// TIA Portal V21 export
FUNCTION "ALARMS PRINT" : Void   // FC2, LAD
{ S7_Optimized_Access := 'TRUE' }
// stored: SetENOAutomatically false
   VAR_TEMP   // added for the SCL form of the ladder/FBD networks
      _w1 : Bool;
      _w2 : Bool;
   END_VAR
BEGIN

REGION Network 1
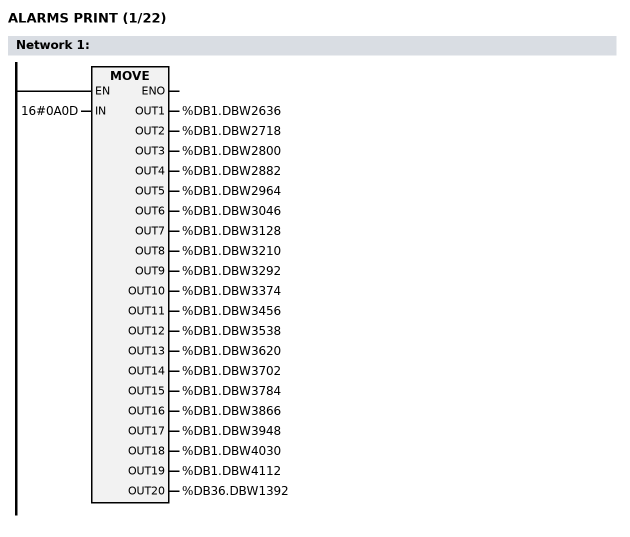
   RUNG wire#powerrail
      Move(in := 16#0A0D, out1 => %DB1.DBW2636, out2 => %DB1.DBW2718, out3 => %DB1.DBW2800, out4 => %DB1.DBW2882, out5 => %DB1.DBW2964, out6 => %DB1.DBW3046, out7 => %DB1.DBW3128, out8 => %DB1.DBW3210, out9 => %DB1.DBW3292, out10 => %DB1.DBW3374, out11 => %DB1.DBW3456, out12 => %DB1.DBW3538, out13 => %DB1.DBW3620, out14 => %DB1.DBW3702, out15 => %DB1.DBW3784, out16 => %DB1.DBW3866, out17 => %DB1.DBW3948, out18 => %DB1.DBW4030, out19 => %DB1.DBW4112, out20 => %DB36.DBW1392)
   END_RUNG
   // the same network as SCL:
   %DB1.DBW2636 := 16#0A0D;
   %DB1.DBW2718 := 16#0A0D;
   %DB1.DBW2800 := 16#0A0D;
   %DB1.DBW2882 := 16#0A0D;
   %DB1.DBW2964 := 16#0A0D;
   %DB1.DBW3046 := 16#0A0D;
   %DB1.DBW3128 := 16#0A0D;
   %DB1.DBW3210 := 16#0A0D;
   %DB1.DBW3292 := 16#0A0D;
   %DB1.DBW3374 := 16#0A0D;
   %DB1.DBW3456 := 16#0A0D;
   %DB1.DBW3538 := 16#0A0D;
   %DB1.DBW3620 := 16#0A0D;
   %DB1.DBW3702 := 16#0A0D;
   %DB1.DBW3784 := 16#0A0D;
   %DB1.DBW3866 := 16#0A0D;
   %DB1.DBW3948 := 16#0A0D;
   %DB1.DBW4030 := 16#0A0D;
   %DB1.DBW4112 := 16#0A0D;
   %DB36.DBW1392 := 16#0A0D;
END_REGION

REGION Network 2
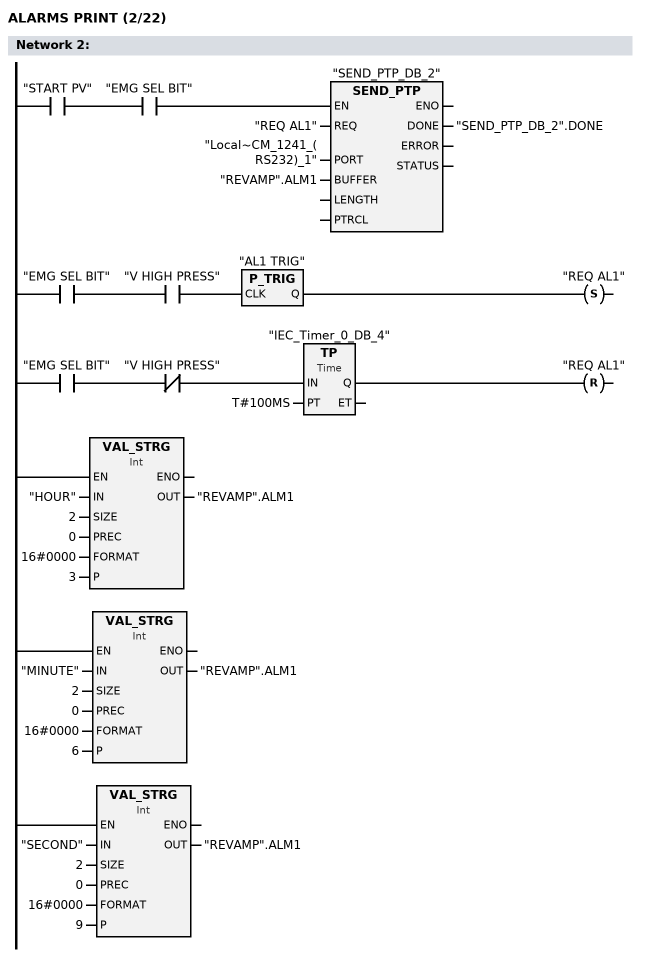
   RUNG wire#powerrail
      Contact( "START PV" )
      Contact( "EMG SEL BIT" )
      "SEND_PTP_DB_2".SEND_PTP(REQ := "REQ AL1", PORT := "Local~CM_1241_(RS232)_1", BUFFER := "REVAMP".ALM1, LENGTH :=, PTRCL :=, DONE => "SEND_PTP_DB_2".DONE, ERROR =>, STATUS =>)
   END_RUNG
   RUNG wire#powerrail
      Contact( "EMG SEL BIT" )
      Contact( "V HIGH PRESS" )
      P_Trig( "AL1 TRIG" )
      S_Coil( "REQ AL1" )
   END_RUNG
   RUNG wire#powerrail
      Contact( "EMG SEL BIT" )
      I_Contact( "V HIGH PRESS" )
      { S7_Templates := "time_type := Time" } "IEC_Timer_0_DB_4".TP(pt := T#100MS, et =>)
      R_Coil( "REQ AL1" )
   END_RUNG
   RUNG wire#powerrail
      { S7_Templates := "[value_type := Int, str_type := String]" } VAL_STRG(IN := "HOUR", SIZE := 2, PREC := 0, FORMAT := 16#0000, P := 3, OUT => "REVAMP".ALM1)
   END_RUNG
   RUNG wire#powerrail
      { S7_Templates := "[value_type := Int, str_type := String]" } VAL_STRG(IN := "MINUTE", SIZE := 2, PREC := 0, FORMAT := 16#0000, P := 6, OUT => "REVAMP".ALM1)
   END_RUNG
   RUNG wire#powerrail
      { S7_Templates := "[value_type := Int, str_type := String]" } VAL_STRG(IN := "SECOND", SIZE := 2, PREC := 0, FORMAT := 16#0000, P := 9, OUT => "REVAMP".ALM1)
   END_RUNG
   // the same network as SCL:
   IF "START PV" AND "EMG SEL BIT" THEN
       "SEND_PTP_DB_2"(REQ := "REQ AL1",   // SEND_PTP
                       PORT := "Local~CM_1241_(RS232)_1",
                       BUFFER := "REVAMP".ALM1,
                       DONE => "SEND_PTP_DB_2".DONE);
   END_IF;
   #_w1 := "EMG SEL BIT" AND "V HIGH PRESS";
   #_w2 := #_w1 AND NOT "AL1 TRIG";   // rising edge
   "AL1 TRIG" := #_w1;
   IF #_w2 THEN "REQ AL1" := TRUE; END_IF;
   "IEC_Timer_0_DB_4".TP(IN := "EMG SEL BIT" AND NOT "V HIGH PRESS", PT := T#100MS);
   IF "IEC_Timer_0_DB_4".Q THEN "REQ AL1" := FALSE; END_IF;
   VAL_STRG(IN := "HOUR", SIZE := 2, PREC := 0, FORMAT := 16#0000, P := 3, OUT => "REVAMP".ALM1);
   VAL_STRG(IN := "MINUTE", SIZE := 2, PREC := 0, FORMAT := 16#0000, P := 6, OUT => "REVAMP".ALM1);
   VAL_STRG(IN := "SECOND", SIZE := 2, PREC := 0, FORMAT := 16#0000, P := 9, OUT => "REVAMP".ALM1);
END_REGION

REGION Network 3
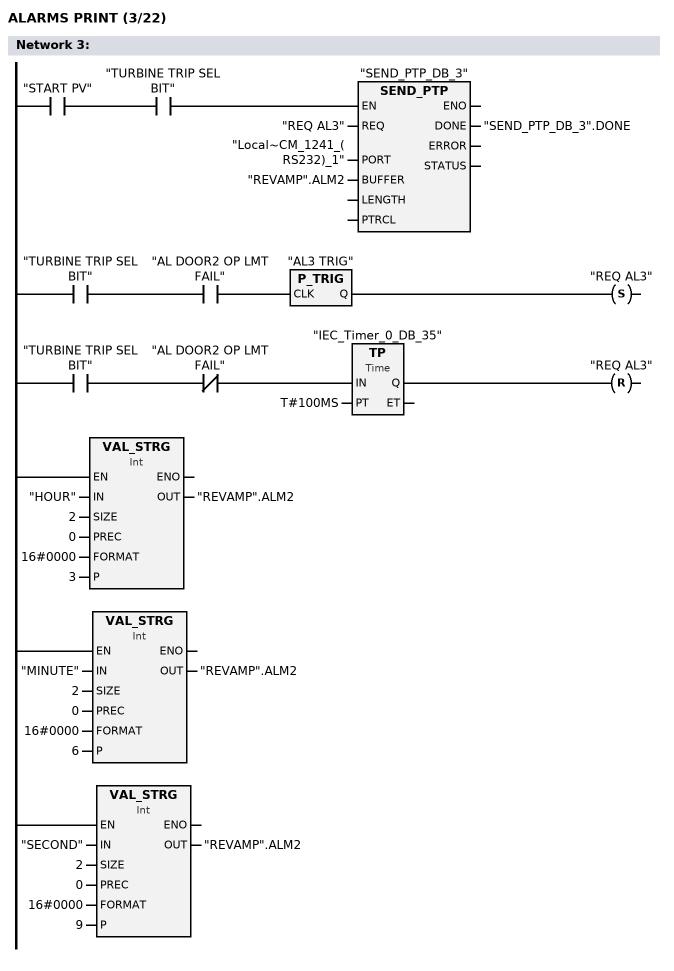
   RUNG wire#powerrail
      Contact( "START PV" )
      Contact( "TURBINE TRIP SEL BIT" )
      "SEND_PTP_DB_3".SEND_PTP(REQ := "REQ AL3", PORT := "Local~CM_1241_(RS232)_1", BUFFER := "REVAMP".ALM2, LENGTH :=, PTRCL :=, DONE => "SEND_PTP_DB_3".DONE, ERROR =>, STATUS =>)
   END_RUNG
   RUNG wire#powerrail
      Contact( "TURBINE TRIP SEL BIT" )
      Contact( "AL DOOR2 OP LMT FAIL" )
      P_Trig( "AL3 TRIG" )
      S_Coil( "REQ AL3" )
   END_RUNG
   RUNG wire#powerrail
      Contact( "TURBINE TRIP SEL BIT" )
      I_Contact( "AL DOOR2 OP LMT FAIL" )
      { S7_Templates := "time_type := Time" } "IEC_Timer_0_DB_35".TP(pt := T#100MS, et =>)
      R_Coil( "REQ AL3" )
   END_RUNG
   RUNG wire#powerrail
      { S7_Templates := "[value_type := Int, str_type := String]" } VAL_STRG(IN := "HOUR", SIZE := 2, PREC := 0, FORMAT := 16#0000, P := 3, OUT => "REVAMP".ALM2)
   END_RUNG
   RUNG wire#powerrail
      { S7_Templates := "[value_type := Int, str_type := String]" } VAL_STRG(IN := "MINUTE", SIZE := 2, PREC := 0, FORMAT := 16#0000, P := 6, OUT => "REVAMP".ALM2)
   END_RUNG
   RUNG wire#powerrail
      { S7_Templates := "[value_type := Int, str_type := String]" } VAL_STRG(IN := "SECOND", SIZE := 2, PREC := 0, FORMAT := 16#0000, P := 9, OUT => "REVAMP".ALM2)
   END_RUNG
   // the same network as SCL:
   IF "START PV" AND "TURBINE TRIP SEL BIT" THEN
       "SEND_PTP_DB_3"(REQ := "REQ AL3",   // SEND_PTP
                       PORT := "Local~CM_1241_(RS232)_1",
                       BUFFER := "REVAMP".ALM2,
                       DONE => "SEND_PTP_DB_3".DONE);
   END_IF;
   #_w1 := "TURBINE TRIP SEL BIT" AND "AL DOOR2 OP LMT FAIL";
   #_w2 := #_w1 AND NOT "AL3 TRIG";   // rising edge
   "AL3 TRIG" := #_w1;
   IF #_w2 THEN "REQ AL3" := TRUE; END_IF;
   "IEC_Timer_0_DB_35".TP(IN := "TURBINE TRIP SEL BIT" AND NOT "AL DOOR2 OP LMT FAIL", PT := T#100MS);
   IF "IEC_Timer_0_DB_35".Q THEN "REQ AL3" := FALSE; END_IF;
   VAL_STRG(IN := "HOUR", SIZE := 2, PREC := 0, FORMAT := 16#0000, P := 3, OUT => "REVAMP".ALM2);
   VAL_STRG(IN := "MINUTE", SIZE := 2, PREC := 0, FORMAT := 16#0000, P := 6, OUT => "REVAMP".ALM2);
   VAL_STRG(IN := "SECOND", SIZE := 2, PREC := 0, FORMAT := 16#0000, P := 9, OUT => "REVAMP".ALM2);
END_REGION

REGION Network 4
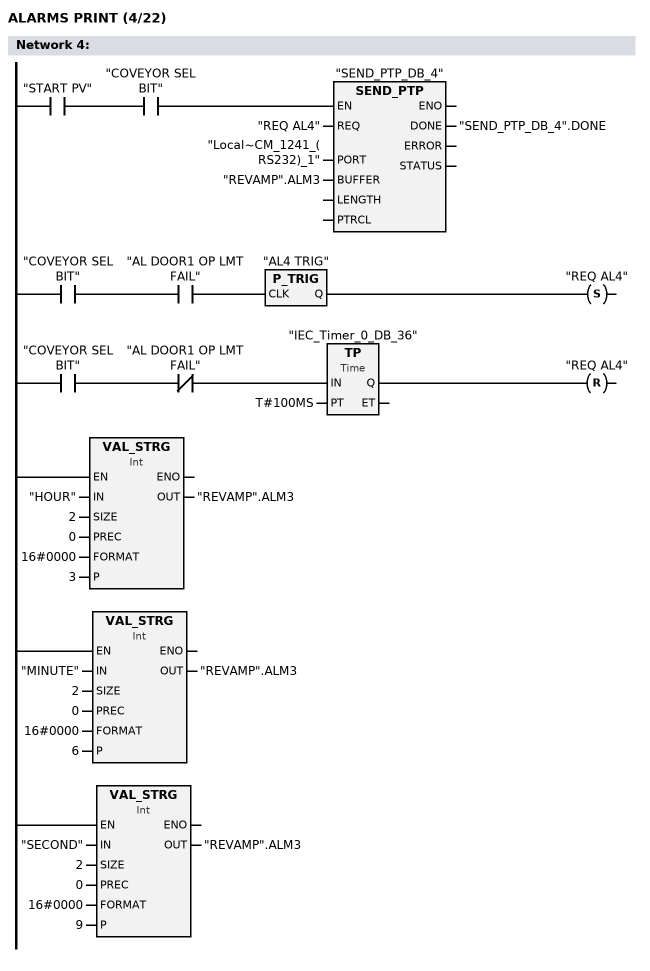
   RUNG wire#powerrail
      Contact( "START PV" )
      Contact( "COVEYOR SEL BIT" )
      "SEND_PTP_DB_4".SEND_PTP(REQ := "REQ AL4", PORT := "Local~CM_1241_(RS232)_1", BUFFER := "REVAMP".ALM3, LENGTH :=, PTRCL :=, DONE => "SEND_PTP_DB_4".DONE, ERROR =>, STATUS =>)
   END_RUNG
   RUNG wire#powerrail
      Contact( "COVEYOR SEL BIT" )
      Contact( "AL DOOR1 OP LMT FAIL" )
      P_Trig( "AL4 TRIG" )
      S_Coil( "REQ AL4" )
   END_RUNG
   RUNG wire#powerrail
      Contact( "COVEYOR SEL BIT" )
      I_Contact( "AL DOOR1 OP LMT FAIL" )
      { S7_Templates := "time_type := Time" } "IEC_Timer_0_DB_36".TP(pt := T#100MS, et =>)
      R_Coil( "REQ AL4" )
   END_RUNG
   RUNG wire#powerrail
      { S7_Templates := "[value_type := Int, str_type := String]" } VAL_STRG(IN := "HOUR", SIZE := 2, PREC := 0, FORMAT := 16#0000, P := 3, OUT => "REVAMP".ALM3)
   END_RUNG
   RUNG wire#powerrail
      { S7_Templates := "[value_type := Int, str_type := String]" } VAL_STRG(IN := "MINUTE", SIZE := 2, PREC := 0, FORMAT := 16#0000, P := 6, OUT => "REVAMP".ALM3)
   END_RUNG
   RUNG wire#powerrail
      { S7_Templates := "[value_type := Int, str_type := String]" } VAL_STRG(IN := "SECOND", SIZE := 2, PREC := 0, FORMAT := 16#0000, P := 9, OUT => "REVAMP".ALM3)
   END_RUNG
   // the same network as SCL:
   IF "START PV" AND "COVEYOR SEL BIT" THEN
       "SEND_PTP_DB_4"(REQ := "REQ AL4",   // SEND_PTP
                       PORT := "Local~CM_1241_(RS232)_1",
                       BUFFER := "REVAMP".ALM3,
                       DONE => "SEND_PTP_DB_4".DONE);
   END_IF;
   #_w1 := "COVEYOR SEL BIT" AND "AL DOOR1 OP LMT FAIL";
   #_w2 := #_w1 AND NOT "AL4 TRIG";   // rising edge
   "AL4 TRIG" := #_w1;
   IF #_w2 THEN "REQ AL4" := TRUE; END_IF;
   "IEC_Timer_0_DB_36".TP(IN := "COVEYOR SEL BIT" AND NOT "AL DOOR1 OP LMT FAIL", PT := T#100MS);
   IF "IEC_Timer_0_DB_36".Q THEN "REQ AL4" := FALSE; END_IF;
   VAL_STRG(IN := "HOUR", SIZE := 2, PREC := 0, FORMAT := 16#0000, P := 3, OUT => "REVAMP".ALM3);
   VAL_STRG(IN := "MINUTE", SIZE := 2, PREC := 0, FORMAT := 16#0000, P := 6, OUT => "REVAMP".ALM3);
   VAL_STRG(IN := "SECOND", SIZE := 2, PREC := 0, FORMAT := 16#0000, P := 9, OUT => "REVAMP".ALM3);
END_REGION

REGION Network 5
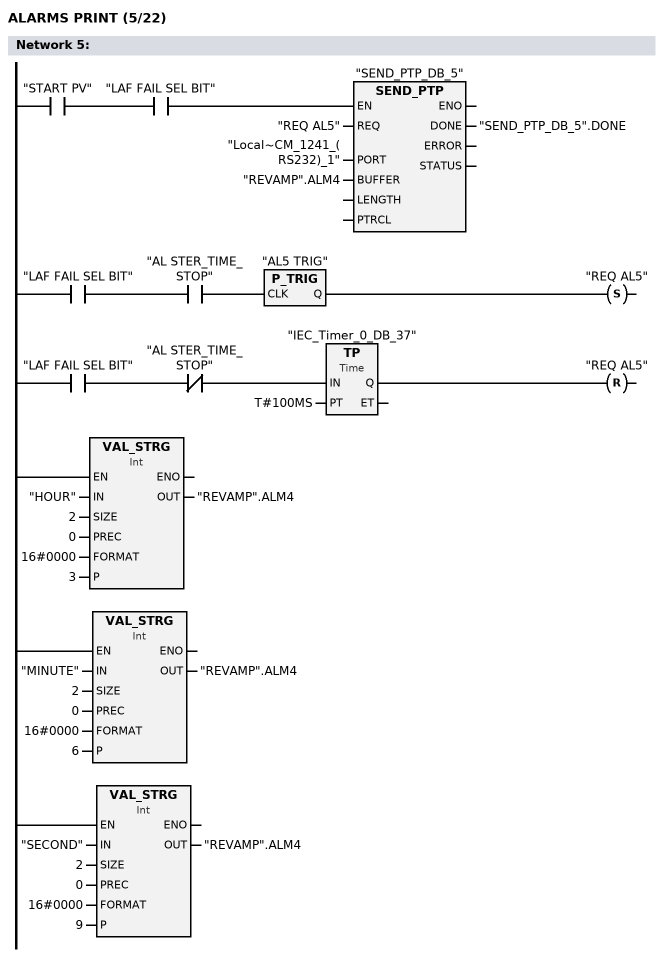
   RUNG wire#powerrail
      Contact( "START PV" )
      Contact( "LAF FAIL SEL BIT" )
      "SEND_PTP_DB_5".SEND_PTP(REQ := "REQ AL5", PORT := "Local~CM_1241_(RS232)_1", BUFFER := "REVAMP".ALM4, LENGTH :=, PTRCL :=, DONE => "SEND_PTP_DB_5".DONE, ERROR =>, STATUS =>)
   END_RUNG
   RUNG wire#powerrail
      Contact( "LAF FAIL SEL BIT" )
      Contact( "AL STER_TIME_STOP" )
      P_Trig( "AL5 TRIG" )
      S_Coil( "REQ AL5" )
   END_RUNG
   RUNG wire#powerrail
      Contact( "LAF FAIL SEL BIT" )
      I_Contact( "AL STER_TIME_STOP" )
      { S7_Templates := "time_type := Time" } "IEC_Timer_0_DB_37".TP(pt := T#100MS, et =>)
      R_Coil( "REQ AL5" )
   END_RUNG
   RUNG wire#powerrail
      { S7_Templates := "[value_type := Int, str_type := String]" } VAL_STRG(IN := "HOUR", SIZE := 2, PREC := 0, FORMAT := 16#0000, P := 3, OUT => "REVAMP".ALM4)
   END_RUNG
   RUNG wire#powerrail
      { S7_Templates := "[value_type := Int, str_type := String]" } VAL_STRG(IN := "MINUTE", SIZE := 2, PREC := 0, FORMAT := 16#0000, P := 6, OUT => "REVAMP".ALM4)
   END_RUNG
   RUNG wire#powerrail
      { S7_Templates := "[value_type := Int, str_type := String]" } VAL_STRG(IN := "SECOND", SIZE := 2, PREC := 0, FORMAT := 16#0000, P := 9, OUT => "REVAMP".ALM4)
   END_RUNG
   // the same network as SCL:
   IF "START PV" AND "LAF FAIL SEL BIT" THEN
       "SEND_PTP_DB_5"(REQ := "REQ AL5",   // SEND_PTP
                       PORT := "Local~CM_1241_(RS232)_1",
                       BUFFER := "REVAMP".ALM4,
                       DONE => "SEND_PTP_DB_5".DONE);
   END_IF;
   #_w1 := "LAF FAIL SEL BIT" AND "AL STER_TIME_STOP";
   #_w2 := #_w1 AND NOT "AL5 TRIG";   // rising edge
   "AL5 TRIG" := #_w1;
   IF #_w2 THEN "REQ AL5" := TRUE; END_IF;
   "IEC_Timer_0_DB_37".TP(IN := "LAF FAIL SEL BIT" AND NOT "AL STER_TIME_STOP", PT := T#100MS);
   IF "IEC_Timer_0_DB_37".Q THEN "REQ AL5" := FALSE; END_IF;
   VAL_STRG(IN := "HOUR", SIZE := 2, PREC := 0, FORMAT := 16#0000, P := 3, OUT => "REVAMP".ALM4);
   VAL_STRG(IN := "MINUTE", SIZE := 2, PREC := 0, FORMAT := 16#0000, P := 6, OUT => "REVAMP".ALM4);
   VAL_STRG(IN := "SECOND", SIZE := 2, PREC := 0, FORMAT := 16#0000, P := 9, OUT => "REVAMP".ALM4);
END_REGION

REGION Network 6
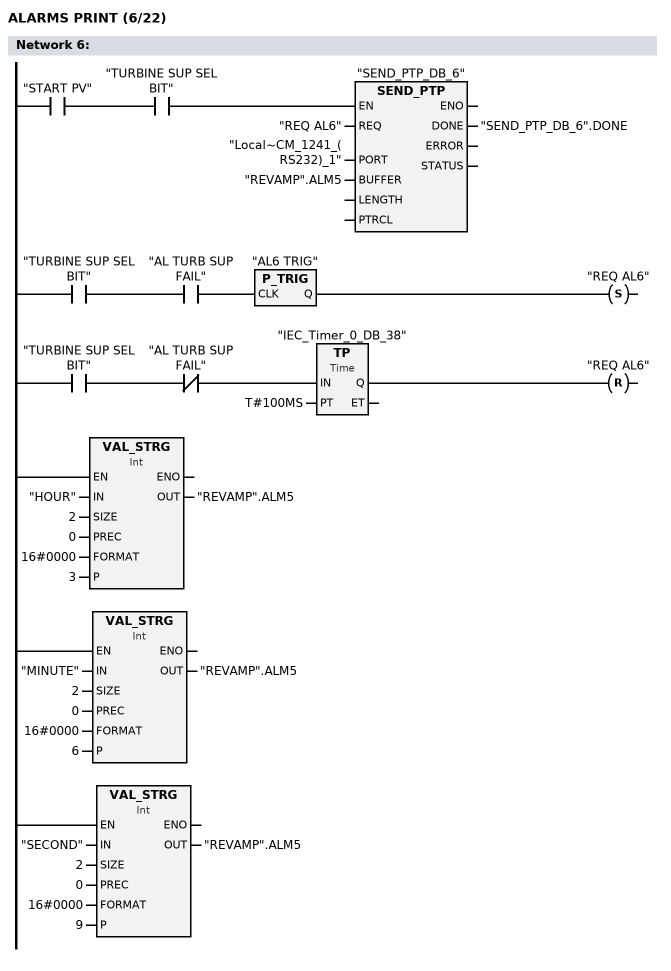
   RUNG wire#powerrail
      Contact( "START PV" )
      Contact( "TURBINE SUP SEL BIT" )
      "SEND_PTP_DB_6".SEND_PTP(REQ := "REQ AL6", PORT := "Local~CM_1241_(RS232)_1", BUFFER := "REVAMP".ALM5, LENGTH :=, PTRCL :=, DONE => "SEND_PTP_DB_6".DONE, ERROR =>, STATUS =>)
   END_RUNG
   RUNG wire#powerrail
      Contact( "TURBINE SUP SEL BIT" )
      Contact( "AL TURB SUP FAIL" )
      P_Trig( "AL6 TRIG" )
      S_Coil( "REQ AL6" )
   END_RUNG
   RUNG wire#powerrail
      Contact( "TURBINE SUP SEL BIT" )
      I_Contact( "AL TURB SUP FAIL" )
      { S7_Templates := "time_type := Time" } "IEC_Timer_0_DB_38".TP(pt := T#100MS, et =>)
      R_Coil( "REQ AL6" )
   END_RUNG
   RUNG wire#powerrail
      { S7_Templates := "[value_type := Int, str_type := String]" } VAL_STRG(IN := "HOUR", SIZE := 2, PREC := 0, FORMAT := 16#0000, P := 3, OUT => "REVAMP".ALM5)
   END_RUNG
   RUNG wire#powerrail
      { S7_Templates := "[value_type := Int, str_type := String]" } VAL_STRG(IN := "MINUTE", SIZE := 2, PREC := 0, FORMAT := 16#0000, P := 6, OUT => "REVAMP".ALM5)
   END_RUNG
   RUNG wire#powerrail
      { S7_Templates := "[value_type := Int, str_type := String]" } VAL_STRG(IN := "SECOND", SIZE := 2, PREC := 0, FORMAT := 16#0000, P := 9, OUT => "REVAMP".ALM5)
   END_RUNG
   // the same network as SCL:
   IF "START PV" AND "TURBINE SUP SEL BIT" THEN
       "SEND_PTP_DB_6"(REQ := "REQ AL6",   // SEND_PTP
                       PORT := "Local~CM_1241_(RS232)_1",
                       BUFFER := "REVAMP".ALM5,
                       DONE => "SEND_PTP_DB_6".DONE);
   END_IF;
   #_w1 := "TURBINE SUP SEL BIT" AND "AL TURB SUP FAIL";
   #_w2 := #_w1 AND NOT "AL6 TRIG";   // rising edge
   "AL6 TRIG" := #_w1;
   IF #_w2 THEN "REQ AL6" := TRUE; END_IF;
   "IEC_Timer_0_DB_38".TP(IN := "TURBINE SUP SEL BIT" AND NOT "AL TURB SUP FAIL", PT := T#100MS);
   IF "IEC_Timer_0_DB_38".Q THEN "REQ AL6" := FALSE; END_IF;
   VAL_STRG(IN := "HOUR", SIZE := 2, PREC := 0, FORMAT := 16#0000, P := 3, OUT => "REVAMP".ALM5);
   VAL_STRG(IN := "MINUTE", SIZE := 2, PREC := 0, FORMAT := 16#0000, P := 6, OUT => "REVAMP".ALM5);
   VAL_STRG(IN := "SECOND", SIZE := 2, PREC := 0, FORMAT := 16#0000, P := 9, OUT => "REVAMP".ALM5);
END_REGION

REGION Network 7
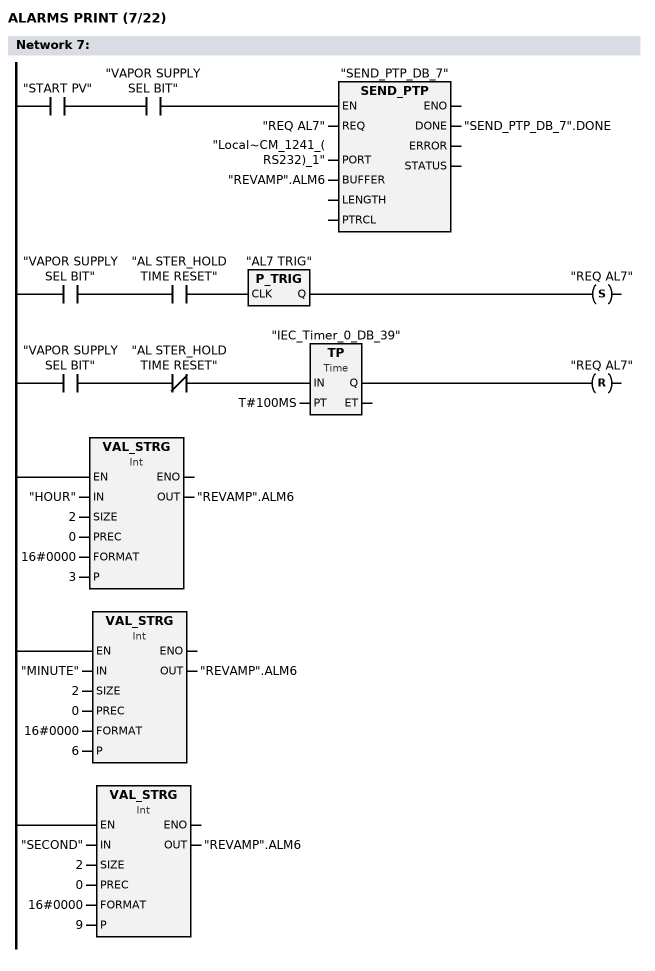
   RUNG wire#powerrail
      Contact( "START PV" )
      Contact( "VAPOR SUPPLY SEL BIT" )
      "SEND_PTP_DB_7".SEND_PTP(REQ := "REQ AL7", PORT := "Local~CM_1241_(RS232)_1", BUFFER := "REVAMP".ALM6, LENGTH :=, PTRCL :=, DONE => "SEND_PTP_DB_7".DONE, ERROR =>, STATUS =>)
   END_RUNG
   RUNG wire#powerrail
      Contact( "VAPOR SUPPLY SEL BIT" )
      Contact( "AL STER_HOLD TIME RESET" )
      P_Trig( "AL7 TRIG" )
      S_Coil( "REQ AL7" )
   END_RUNG
   RUNG wire#powerrail
      Contact( "VAPOR SUPPLY SEL BIT" )
      I_Contact( "AL STER_HOLD TIME RESET" )
      { S7_Templates := "time_type := Time" } "IEC_Timer_0_DB_39".TP(pt := T#100MS, et =>)
      R_Coil( "REQ AL7" )
   END_RUNG
   RUNG wire#powerrail
      { S7_Templates := "[value_type := Int, str_type := String]" } VAL_STRG(IN := "HOUR", SIZE := 2, PREC := 0, FORMAT := 16#0000, P := 3, OUT => "REVAMP".ALM6)
   END_RUNG
   RUNG wire#powerrail
      { S7_Templates := "[value_type := Int, str_type := String]" } VAL_STRG(IN := "MINUTE", SIZE := 2, PREC := 0, FORMAT := 16#0000, P := 6, OUT => "REVAMP".ALM6)
   END_RUNG
   RUNG wire#powerrail
      { S7_Templates := "[value_type := Int, str_type := String]" } VAL_STRG(IN := "SECOND", SIZE := 2, PREC := 0, FORMAT := 16#0000, P := 9, OUT => "REVAMP".ALM6)
   END_RUNG
   // the same network as SCL:
   IF "START PV" AND "VAPOR SUPPLY SEL BIT" THEN
       "SEND_PTP_DB_7"(REQ := "REQ AL7",   // SEND_PTP
                       PORT := "Local~CM_1241_(RS232)_1",
                       BUFFER := "REVAMP".ALM6,
                       DONE => "SEND_PTP_DB_7".DONE);
   END_IF;
   #_w1 := "VAPOR SUPPLY SEL BIT" AND "AL STER_HOLD TIME RESET";
   #_w2 := #_w1 AND NOT "AL7 TRIG";   // rising edge
   "AL7 TRIG" := #_w1;
   IF #_w2 THEN "REQ AL7" := TRUE; END_IF;
   "IEC_Timer_0_DB_39".TP(IN := "VAPOR SUPPLY SEL BIT" AND NOT "AL STER_HOLD TIME RESET", PT := T#100MS);
   IF "IEC_Timer_0_DB_39".Q THEN "REQ AL7" := FALSE; END_IF;
   VAL_STRG(IN := "HOUR", SIZE := 2, PREC := 0, FORMAT := 16#0000, P := 3, OUT => "REVAMP".ALM6);
   VAL_STRG(IN := "MINUTE", SIZE := 2, PREC := 0, FORMAT := 16#0000, P := 6, OUT => "REVAMP".ALM6);
   VAL_STRG(IN := "SECOND", SIZE := 2, PREC := 0, FORMAT := 16#0000, P := 9, OUT => "REVAMP".ALM6);
END_REGION

REGION Network 8
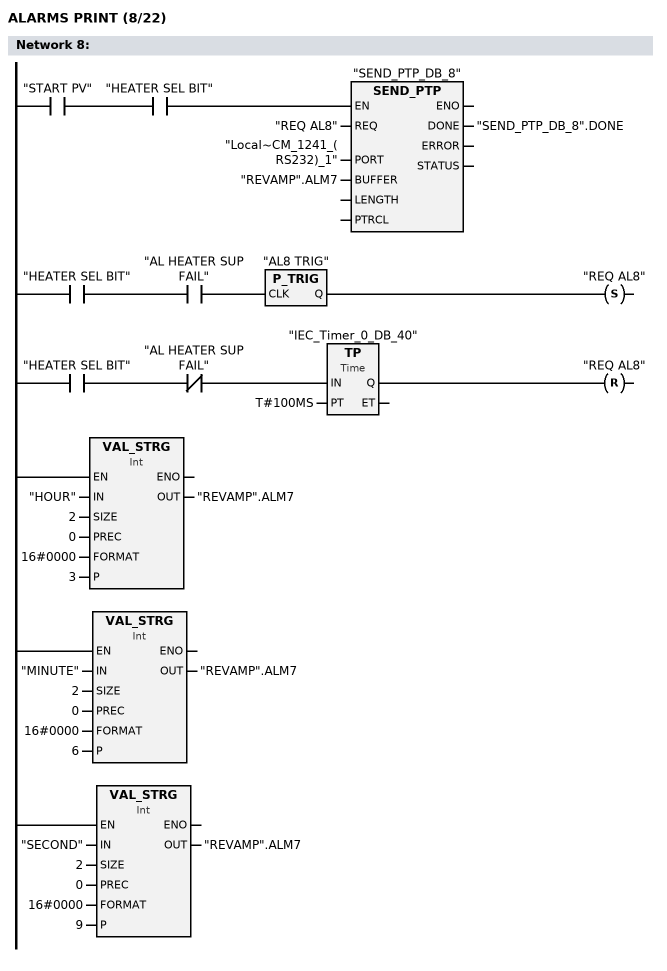
   RUNG wire#powerrail
      Contact( "START PV" )
      Contact( "HEATER SEL BIT" )
      "SEND_PTP_DB_8".SEND_PTP(REQ := "REQ AL8", PORT := "Local~CM_1241_(RS232)_1", BUFFER := "REVAMP".ALM7, LENGTH :=, PTRCL :=, DONE => "SEND_PTP_DB_8".DONE, ERROR =>, STATUS =>)
   END_RUNG
   RUNG wire#powerrail
      Contact( "HEATER SEL BIT" )
      Contact( "AL HEATER SUP FAIL" )
      P_Trig( "AL8 TRIG" )
      S_Coil( "REQ AL8" )
   END_RUNG
   RUNG wire#powerrail
      Contact( "HEATER SEL BIT" )
      I_Contact( "AL HEATER SUP FAIL" )
      { S7_Templates := "time_type := Time" } "IEC_Timer_0_DB_40".TP(pt := T#100MS, et =>)
      R_Coil( "REQ AL8" )
   END_RUNG
   RUNG wire#powerrail
      { S7_Templates := "[value_type := Int, str_type := String]" } VAL_STRG(IN := "HOUR", SIZE := 2, PREC := 0, FORMAT := 16#0000, P := 3, OUT => "REVAMP".ALM7)
   END_RUNG
   RUNG wire#powerrail
      { S7_Templates := "[value_type := Int, str_type := String]" } VAL_STRG(IN := "MINUTE", SIZE := 2, PREC := 0, FORMAT := 16#0000, P := 6, OUT => "REVAMP".ALM7)
   END_RUNG
   RUNG wire#powerrail
      { S7_Templates := "[value_type := Int, str_type := String]" } VAL_STRG(IN := "SECOND", SIZE := 2, PREC := 0, FORMAT := 16#0000, P := 9, OUT => "REVAMP".ALM7)
   END_RUNG
   // the same network as SCL:
   IF "START PV" AND "HEATER SEL BIT" THEN
       "SEND_PTP_DB_8"(REQ := "REQ AL8",   // SEND_PTP
                       PORT := "Local~CM_1241_(RS232)_1",
                       BUFFER := "REVAMP".ALM7,
                       DONE => "SEND_PTP_DB_8".DONE);
   END_IF;
   #_w1 := "HEATER SEL BIT" AND "AL HEATER SUP FAIL";
   #_w2 := #_w1 AND NOT "AL8 TRIG";   // rising edge
   "AL8 TRIG" := #_w1;
   IF #_w2 THEN "REQ AL8" := TRUE; END_IF;
   "IEC_Timer_0_DB_40".TP(IN := "HEATER SEL BIT" AND NOT "AL HEATER SUP FAIL", PT := T#100MS);
   IF "IEC_Timer_0_DB_40".Q THEN "REQ AL8" := FALSE; END_IF;
   VAL_STRG(IN := "HOUR", SIZE := 2, PREC := 0, FORMAT := 16#0000, P := 3, OUT => "REVAMP".ALM7);
   VAL_STRG(IN := "MINUTE", SIZE := 2, PREC := 0, FORMAT := 16#0000, P := 6, OUT => "REVAMP".ALM7);
   VAL_STRG(IN := "SECOND", SIZE := 2, PREC := 0, FORMAT := 16#0000, P := 9, OUT => "REVAMP".ALM7);
END_REGION

REGION Network 9
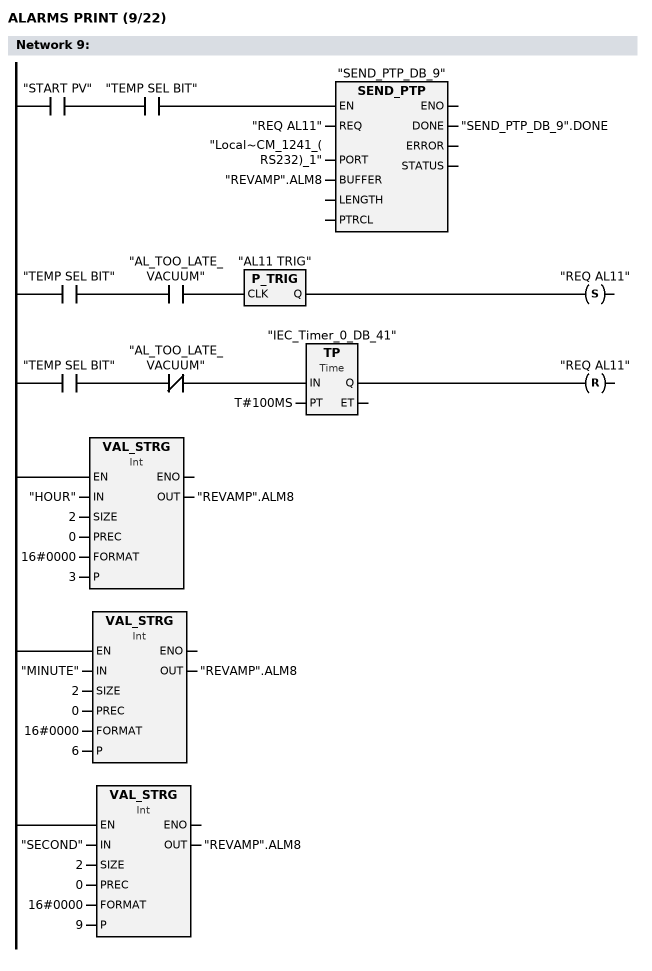
   RUNG wire#powerrail
      Contact( "START PV" )
      Contact( "TEMP SEL BIT" )
      "SEND_PTP_DB_9".SEND_PTP(REQ := "REQ AL11", PORT := "Local~CM_1241_(RS232)_1", BUFFER := "REVAMP".ALM8, LENGTH :=, PTRCL :=, DONE => "SEND_PTP_DB_9".DONE, ERROR =>, STATUS =>)
   END_RUNG
   RUNG wire#powerrail
      Contact( "TEMP SEL BIT" )
      Contact( "AL_TOO_LATE_VACUUM" )
      P_Trig( "AL11 TRIG" )
      S_Coil( "REQ AL11" )
   END_RUNG
   RUNG wire#powerrail
      Contact( "TEMP SEL BIT" )
      I_Contact( "AL_TOO_LATE_VACUUM" )
      { S7_Templates := "time_type := Time" } "IEC_Timer_0_DB_41".TP(pt := T#100MS, et =>)
      R_Coil( "REQ AL11" )
   END_RUNG
   RUNG wire#powerrail
      { S7_Templates := "[value_type := Int, str_type := String]" } VAL_STRG(IN := "HOUR", SIZE := 2, PREC := 0, FORMAT := 16#0000, P := 3, OUT => "REVAMP".ALM8)
   END_RUNG
   RUNG wire#powerrail
      { S7_Templates := "[value_type := Int, str_type := String]" } VAL_STRG(IN := "MINUTE", SIZE := 2, PREC := 0, FORMAT := 16#0000, P := 6, OUT => "REVAMP".ALM8)
   END_RUNG
   RUNG wire#powerrail
      { S7_Templates := "[value_type := Int, str_type := String]" } VAL_STRG(IN := "SECOND", SIZE := 2, PREC := 0, FORMAT := 16#0000, P := 9, OUT => "REVAMP".ALM8)
   END_RUNG
   // the same network as SCL:
   IF "START PV" AND "TEMP SEL BIT" THEN
       "SEND_PTP_DB_9"(REQ := "REQ AL11",   // SEND_PTP
                       PORT := "Local~CM_1241_(RS232)_1",
                       BUFFER := "REVAMP".ALM8,
                       DONE => "SEND_PTP_DB_9".DONE);
   END_IF;
   #_w1 := "TEMP SEL BIT" AND "AL_TOO_LATE_VACUUM";
   #_w2 := #_w1 AND NOT "AL11 TRIG";   // rising edge
   "AL11 TRIG" := #_w1;
   IF #_w2 THEN "REQ AL11" := TRUE; END_IF;
   "IEC_Timer_0_DB_41".TP(IN := "TEMP SEL BIT" AND NOT "AL_TOO_LATE_VACUUM", PT := T#100MS);
   IF "IEC_Timer_0_DB_41".Q THEN "REQ AL11" := FALSE; END_IF;
   VAL_STRG(IN := "HOUR", SIZE := 2, PREC := 0, FORMAT := 16#0000, P := 3, OUT => "REVAMP".ALM8);
   VAL_STRG(IN := "MINUTE", SIZE := 2, PREC := 0, FORMAT := 16#0000, P := 6, OUT => "REVAMP".ALM8);
   VAL_STRG(IN := "SECOND", SIZE := 2, PREC := 0, FORMAT := 16#0000, P := 9, OUT => "REVAMP".ALM8);
END_REGION

REGION Network 10
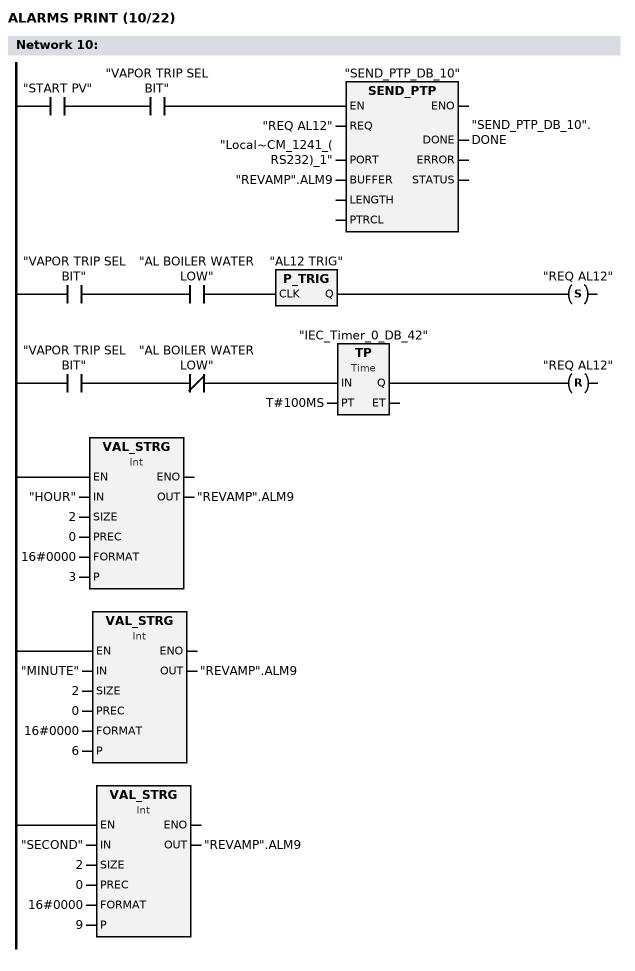
   RUNG wire#powerrail
      Contact( "START PV" )
      Contact( "VAPOR TRIP SEL BIT" )
      "SEND_PTP_DB_10".SEND_PTP(REQ := "REQ AL12", PORT := "Local~CM_1241_(RS232)_1", BUFFER := "REVAMP".ALM9, LENGTH :=, PTRCL :=, DONE => "SEND_PTP_DB_10".DONE, ERROR =>, STATUS =>)
   END_RUNG
   RUNG wire#powerrail
      Contact( "VAPOR TRIP SEL BIT" )
      Contact( "AL BOILER WATER LOW" )
      P_Trig( "AL12 TRIG" )
      S_Coil( "REQ AL12" )
   END_RUNG
   RUNG wire#powerrail
      Contact( "VAPOR TRIP SEL BIT" )
      I_Contact( "AL BOILER WATER LOW" )
      { S7_Templates := "time_type := Time" } "IEC_Timer_0_DB_42".TP(pt := T#100MS, et =>)
      R_Coil( "REQ AL12" )
   END_RUNG
   RUNG wire#powerrail
      { S7_Templates := "[value_type := Int, str_type := String]" } VAL_STRG(IN := "HOUR", SIZE := 2, PREC := 0, FORMAT := 16#0000, P := 3, OUT => "REVAMP".ALM9)
   END_RUNG
   RUNG wire#powerrail
      { S7_Templates := "[value_type := Int, str_type := String]" } VAL_STRG(IN := "MINUTE", SIZE := 2, PREC := 0, FORMAT := 16#0000, P := 6, OUT => "REVAMP".ALM9)
   END_RUNG
   RUNG wire#powerrail
      { S7_Templates := "[value_type := Int, str_type := String]" } VAL_STRG(IN := "SECOND", SIZE := 2, PREC := 0, FORMAT := 16#0000, P := 9, OUT => "REVAMP".ALM9)
   END_RUNG
   // the same network as SCL:
   IF "START PV" AND "VAPOR TRIP SEL BIT" THEN
       "SEND_PTP_DB_10"(REQ := "REQ AL12",   // SEND_PTP
                        PORT := "Local~CM_1241_(RS232)_1",
                        BUFFER := "REVAMP".ALM9,
                        DONE => "SEND_PTP_DB_10".DONE);
   END_IF;
   #_w1 := "VAPOR TRIP SEL BIT" AND "AL BOILER WATER LOW";
   #_w2 := #_w1 AND NOT "AL12 TRIG";   // rising edge
   "AL12 TRIG" := #_w1;
   IF #_w2 THEN "REQ AL12" := TRUE; END_IF;
   "IEC_Timer_0_DB_42".TP(IN := "VAPOR TRIP SEL BIT" AND NOT "AL BOILER WATER LOW", PT := T#100MS);
   IF "IEC_Timer_0_DB_42".Q THEN "REQ AL12" := FALSE; END_IF;
   VAL_STRG(IN := "HOUR", SIZE := 2, PREC := 0, FORMAT := 16#0000, P := 3, OUT => "REVAMP".ALM9);
   VAL_STRG(IN := "MINUTE", SIZE := 2, PREC := 0, FORMAT := 16#0000, P := 6, OUT => "REVAMP".ALM9);
   VAL_STRG(IN := "SECOND", SIZE := 2, PREC := 0, FORMAT := 16#0000, P := 9, OUT => "REVAMP".ALM9);
END_REGION

REGION Network 11
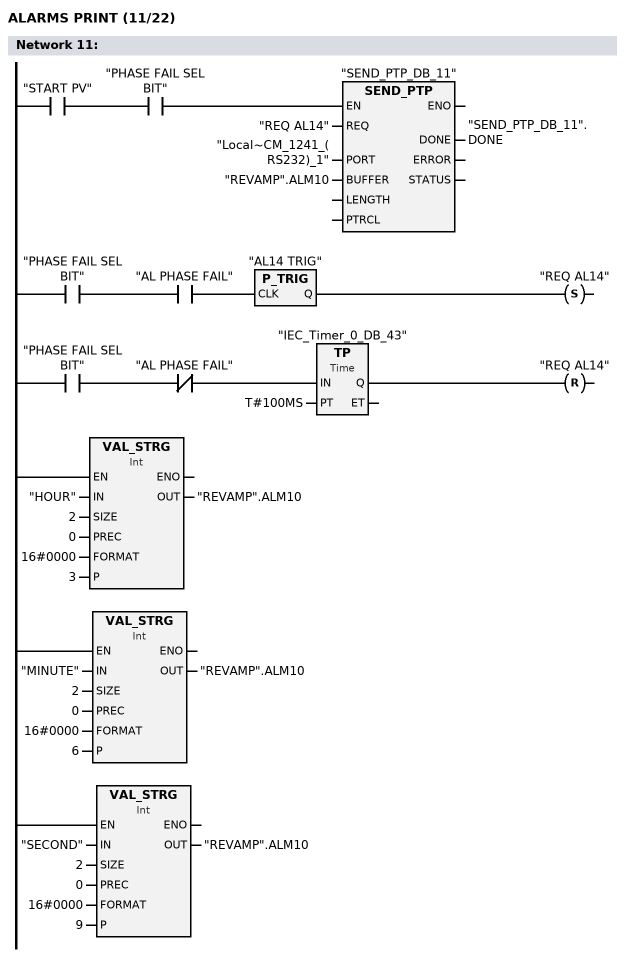
   RUNG wire#powerrail
      Contact( "START PV" )
      Contact( "PHASE FAIL SEL BIT" )
      "SEND_PTP_DB_11".SEND_PTP(REQ := "REQ AL14", PORT := "Local~CM_1241_(RS232)_1", BUFFER := "REVAMP".ALM10, LENGTH :=, PTRCL :=, DONE => "SEND_PTP_DB_11".DONE, ERROR =>, STATUS =>)
   END_RUNG
   RUNG wire#powerrail
      Contact( "PHASE FAIL SEL BIT" )
      Contact( "AL PHASE FAIL" )
      P_Trig( "AL14 TRIG" )
      S_Coil( "REQ AL14" )
   END_RUNG
   RUNG wire#powerrail
      Contact( "PHASE FAIL SEL BIT" )
      I_Contact( "AL PHASE FAIL" )
      { S7_Templates := "time_type := Time" } "IEC_Timer_0_DB_43".TP(pt := T#100MS, et =>)
      R_Coil( "REQ AL14" )
   END_RUNG
   RUNG wire#powerrail
      { S7_Templates := "[value_type := Int, str_type := String]" } VAL_STRG(IN := "HOUR", SIZE := 2, PREC := 0, FORMAT := 16#0000, P := 3, OUT => "REVAMP".ALM10)
   END_RUNG
   RUNG wire#powerrail
      { S7_Templates := "[value_type := Int, str_type := String]" } VAL_STRG(IN := "MINUTE", SIZE := 2, PREC := 0, FORMAT := 16#0000, P := 6, OUT => "REVAMP".ALM10)
   END_RUNG
   RUNG wire#powerrail
      { S7_Templates := "[value_type := Int, str_type := String]" } VAL_STRG(IN := "SECOND", SIZE := 2, PREC := 0, FORMAT := 16#0000, P := 9, OUT => "REVAMP".ALM10)
   END_RUNG
   // the same network as SCL:
   IF "START PV" AND "PHASE FAIL SEL BIT" THEN
       "SEND_PTP_DB_11"(REQ := "REQ AL14",   // SEND_PTP
                        PORT := "Local~CM_1241_(RS232)_1",
                        BUFFER := "REVAMP".ALM10,
                        DONE => "SEND_PTP_DB_11".DONE);
   END_IF;
   #_w1 := "PHASE FAIL SEL BIT" AND "AL PHASE FAIL";
   #_w2 := #_w1 AND NOT "AL14 TRIG";   // rising edge
   "AL14 TRIG" := #_w1;
   IF #_w2 THEN "REQ AL14" := TRUE; END_IF;
   "IEC_Timer_0_DB_43".TP(IN := "PHASE FAIL SEL BIT" AND NOT "AL PHASE FAIL", PT := T#100MS);
   IF "IEC_Timer_0_DB_43".Q THEN "REQ AL14" := FALSE; END_IF;
   VAL_STRG(IN := "HOUR", SIZE := 2, PREC := 0, FORMAT := 16#0000, P := 3, OUT => "REVAMP".ALM10);
   VAL_STRG(IN := "MINUTE", SIZE := 2, PREC := 0, FORMAT := 16#0000, P := 6, OUT => "REVAMP".ALM10);
   VAL_STRG(IN := "SECOND", SIZE := 2, PREC := 0, FORMAT := 16#0000, P := 9, OUT => "REVAMP".ALM10);
END_REGION

REGION Network 12
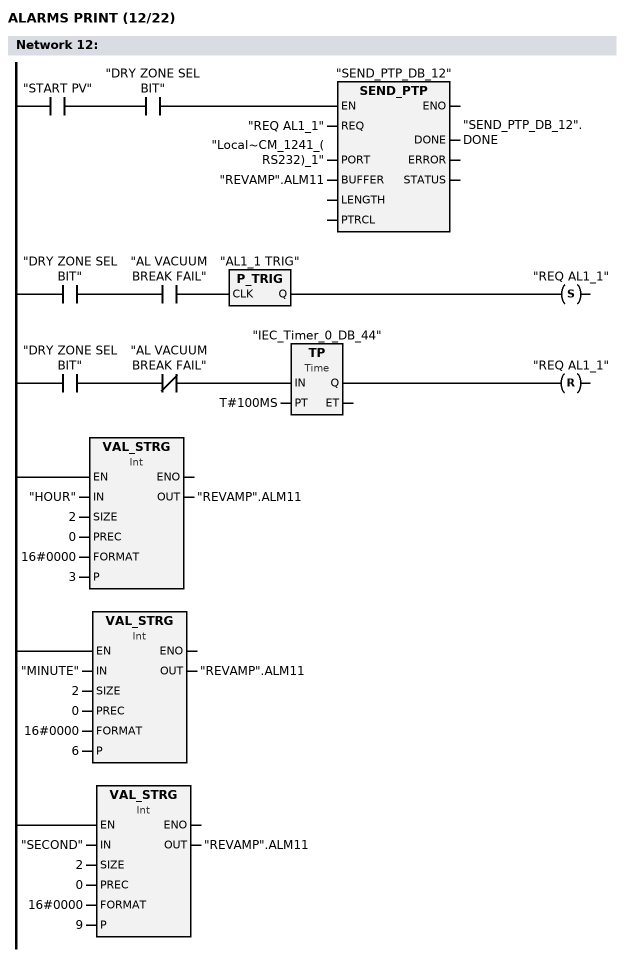
   RUNG wire#powerrail
      Contact( "START PV" )
      Contact( "DRY ZONE SEL BIT" )
      "SEND_PTP_DB_12".SEND_PTP(REQ := "REQ AL1_1", PORT := "Local~CM_1241_(RS232)_1", BUFFER := "REVAMP".ALM11, LENGTH :=, PTRCL :=, DONE => "SEND_PTP_DB_12".DONE, ERROR =>, STATUS =>)
   END_RUNG
   RUNG wire#powerrail
      Contact( "DRY ZONE SEL BIT" )
      Contact( "AL VACUUM BREAK FAIL" )
      P_Trig( "AL1_1 TRIG" )
      S_Coil( "REQ AL1_1" )
   END_RUNG
   RUNG wire#powerrail
      Contact( "DRY ZONE SEL BIT" )
      I_Contact( "AL VACUUM BREAK FAIL" )
      { S7_Templates := "time_type := Time" } "IEC_Timer_0_DB_44".TP(pt := T#100MS, et =>)
      R_Coil( "REQ AL1_1" )
   END_RUNG
   RUNG wire#powerrail
      { S7_Templates := "[value_type := Int, str_type := String]" } VAL_STRG(IN := "HOUR", SIZE := 2, PREC := 0, FORMAT := 16#0000, P := 3, OUT => "REVAMP".ALM11)
   END_RUNG
   RUNG wire#powerrail
      { S7_Templates := "[value_type := Int, str_type := String]" } VAL_STRG(IN := "MINUTE", SIZE := 2, PREC := 0, FORMAT := 16#0000, P := 6, OUT => "REVAMP".ALM11)
   END_RUNG
   RUNG wire#powerrail
      { S7_Templates := "[value_type := Int, str_type := String]" } VAL_STRG(IN := "SECOND", SIZE := 2, PREC := 0, FORMAT := 16#0000, P := 9, OUT => "REVAMP".ALM11)
   END_RUNG
   // the same network as SCL:
   IF "START PV" AND "DRY ZONE SEL BIT" THEN
       "SEND_PTP_DB_12"(REQ := "REQ AL1_1",   // SEND_PTP
                        PORT := "Local~CM_1241_(RS232)_1",
                        BUFFER := "REVAMP".ALM11,
                        DONE => "SEND_PTP_DB_12".DONE);
   END_IF;
   #_w1 := "DRY ZONE SEL BIT" AND "AL VACUUM BREAK FAIL";
   #_w2 := #_w1 AND NOT "AL1_1 TRIG";   // rising edge
   "AL1_1 TRIG" := #_w1;
   IF #_w2 THEN "REQ AL1_1" := TRUE; END_IF;
   "IEC_Timer_0_DB_44".TP(IN := "DRY ZONE SEL BIT" AND NOT "AL VACUUM BREAK FAIL", PT := T#100MS);
   IF "IEC_Timer_0_DB_44".Q THEN "REQ AL1_1" := FALSE; END_IF;
   VAL_STRG(IN := "HOUR", SIZE := 2, PREC := 0, FORMAT := 16#0000, P := 3, OUT => "REVAMP".ALM11);
   VAL_STRG(IN := "MINUTE", SIZE := 2, PREC := 0, FORMAT := 16#0000, P := 6, OUT => "REVAMP".ALM11);
   VAL_STRG(IN := "SECOND", SIZE := 2, PREC := 0, FORMAT := 16#0000, P := 9, OUT => "REVAMP".ALM11);
END_REGION

REGION Network 13
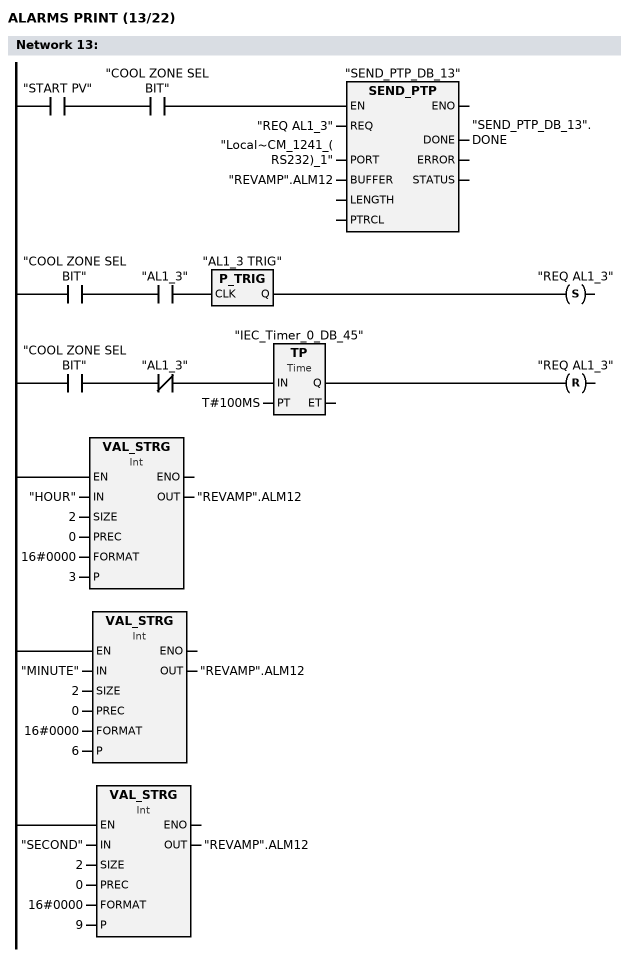
   RUNG wire#powerrail
      Contact( "START PV" )
      Contact( "COOL ZONE SEL BIT" )
      "SEND_PTP_DB_13".SEND_PTP(REQ := "REQ AL1_3", PORT := "Local~CM_1241_(RS232)_1", BUFFER := "REVAMP".ALM12, LENGTH :=, PTRCL :=, DONE => "SEND_PTP_DB_13".DONE, ERROR =>, STATUS =>)
   END_RUNG
   RUNG wire#powerrail
      Contact( "COOL ZONE SEL BIT" )
      Contact( "AL1_3" )
      P_Trig( "AL1_3 TRIG" )
      S_Coil( "REQ AL1_3" )
   END_RUNG
   RUNG wire#powerrail
      Contact( "COOL ZONE SEL BIT" )
      I_Contact( "AL1_3" )
      { S7_Templates := "time_type := Time" } "IEC_Timer_0_DB_45".TP(pt := T#100MS, et =>)
      R_Coil( "REQ AL1_3" )
   END_RUNG
   RUNG wire#powerrail
      { S7_Templates := "[value_type := Int, str_type := String]" } VAL_STRG(IN := "HOUR", SIZE := 2, PREC := 0, FORMAT := 16#0000, P := 3, OUT => "REVAMP".ALM12)
   END_RUNG
   RUNG wire#powerrail
      { S7_Templates := "[value_type := Int, str_type := String]" } VAL_STRG(IN := "MINUTE", SIZE := 2, PREC := 0, FORMAT := 16#0000, P := 6, OUT => "REVAMP".ALM12)
   END_RUNG
   RUNG wire#powerrail
      { S7_Templates := "[value_type := Int, str_type := String]" } VAL_STRG(IN := "SECOND", SIZE := 2, PREC := 0, FORMAT := 16#0000, P := 9, OUT => "REVAMP".ALM12)
   END_RUNG
   // the same network as SCL:
   IF "START PV" AND "COOL ZONE SEL BIT" THEN
       "SEND_PTP_DB_13"(REQ := "REQ AL1_3",   // SEND_PTP
                        PORT := "Local~CM_1241_(RS232)_1",
                        BUFFER := "REVAMP".ALM12,
                        DONE => "SEND_PTP_DB_13".DONE);
   END_IF;
   #_w1 := "COOL ZONE SEL BIT" AND "AL1_3";
   #_w2 := #_w1 AND NOT "AL1_3 TRIG";   // rising edge
   "AL1_3 TRIG" := #_w1;
   IF #_w2 THEN "REQ AL1_3" := TRUE; END_IF;
   "IEC_Timer_0_DB_45".TP(IN := "COOL ZONE SEL BIT" AND NOT "AL1_3", PT := T#100MS);
   IF "IEC_Timer_0_DB_45".Q THEN "REQ AL1_3" := FALSE; END_IF;
   VAL_STRG(IN := "HOUR", SIZE := 2, PREC := 0, FORMAT := 16#0000, P := 3, OUT => "REVAMP".ALM12);
   VAL_STRG(IN := "MINUTE", SIZE := 2, PREC := 0, FORMAT := 16#0000, P := 6, OUT => "REVAMP".ALM12);
   VAL_STRG(IN := "SECOND", SIZE := 2, PREC := 0, FORMAT := 16#0000, P := 9, OUT => "REVAMP".ALM12);
END_REGION

REGION Network 14
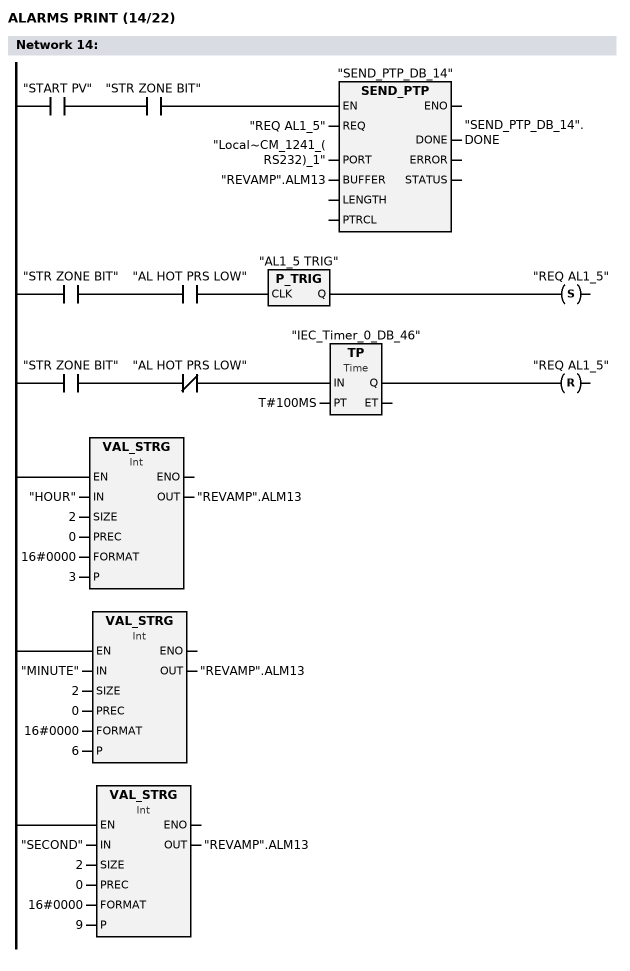
   RUNG wire#powerrail
      Contact( "START PV" )
      Contact( "STR ZONE BIT" )
      "SEND_PTP_DB_14".SEND_PTP(REQ := "REQ AL1_5", PORT := "Local~CM_1241_(RS232)_1", BUFFER := "REVAMP".ALM13, LENGTH :=, PTRCL :=, DONE => "SEND_PTP_DB_14".DONE, ERROR =>, STATUS =>)
   END_RUNG
   RUNG wire#powerrail
      Contact( "STR ZONE BIT" )
      Contact( "AL HOT PRS LOW" )
      P_Trig( "AL1_5 TRIG" )
      S_Coil( "REQ AL1_5" )
   END_RUNG
   RUNG wire#powerrail
      Contact( "STR ZONE BIT" )
      I_Contact( "AL HOT PRS LOW" )
      { S7_Templates := "time_type := Time" } "IEC_Timer_0_DB_46".TP(pt := T#100MS, et =>)
      R_Coil( "REQ AL1_5" )
   END_RUNG
   RUNG wire#powerrail
      { S7_Templates := "[value_type := Int, str_type := String]" } VAL_STRG(IN := "HOUR", SIZE := 2, PREC := 0, FORMAT := 16#0000, P := 3, OUT => "REVAMP".ALM13)
   END_RUNG
   RUNG wire#powerrail
      { S7_Templates := "[value_type := Int, str_type := String]" } VAL_STRG(IN := "MINUTE", SIZE := 2, PREC := 0, FORMAT := 16#0000, P := 6, OUT => "REVAMP".ALM13)
   END_RUNG
   RUNG wire#powerrail
      { S7_Templates := "[value_type := Int, str_type := String]" } VAL_STRG(IN := "SECOND", SIZE := 2, PREC := 0, FORMAT := 16#0000, P := 9, OUT => "REVAMP".ALM13)
   END_RUNG
   // the same network as SCL:
   IF "START PV" AND "STR ZONE BIT" THEN
       "SEND_PTP_DB_14"(REQ := "REQ AL1_5",   // SEND_PTP
                        PORT := "Local~CM_1241_(RS232)_1",
                        BUFFER := "REVAMP".ALM13,
                        DONE => "SEND_PTP_DB_14".DONE);
   END_IF;
   #_w1 := "STR ZONE BIT" AND "AL HOT PRS LOW";
   #_w2 := #_w1 AND NOT "AL1_5 TRIG";   // rising edge
   "AL1_5 TRIG" := #_w1;
   IF #_w2 THEN "REQ AL1_5" := TRUE; END_IF;
   "IEC_Timer_0_DB_46".TP(IN := "STR ZONE BIT" AND NOT "AL HOT PRS LOW", PT := T#100MS);
   IF "IEC_Timer_0_DB_46".Q THEN "REQ AL1_5" := FALSE; END_IF;
   VAL_STRG(IN := "HOUR", SIZE := 2, PREC := 0, FORMAT := 16#0000, P := 3, OUT => "REVAMP".ALM13);
   VAL_STRG(IN := "MINUTE", SIZE := 2, PREC := 0, FORMAT := 16#0000, P := 6, OUT => "REVAMP".ALM13);
   VAL_STRG(IN := "SECOND", SIZE := 2, PREC := 0, FORMAT := 16#0000, P := 9, OUT => "REVAMP".ALM13);
END_REGION

REGION Network 15
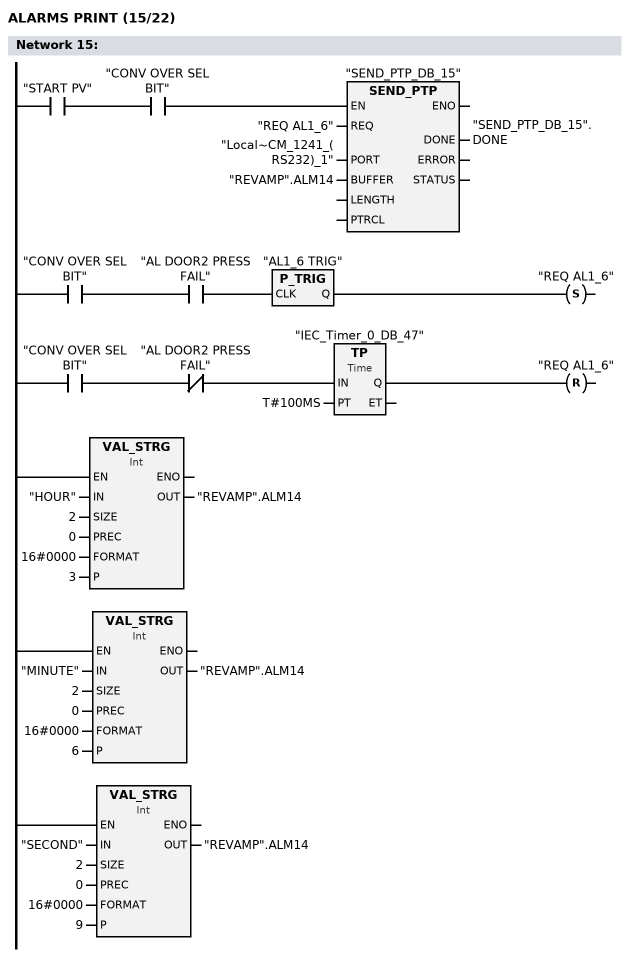
   RUNG wire#powerrail
      Contact( "START PV" )
      Contact( "CONV OVER SEL BIT" )
      "SEND_PTP_DB_15".SEND_PTP(REQ := "REQ AL1_6", PORT := "Local~CM_1241_(RS232)_1", BUFFER := "REVAMP".ALM14, LENGTH :=, PTRCL :=, DONE => "SEND_PTP_DB_15".DONE, ERROR =>, STATUS =>)
   END_RUNG
   RUNG wire#powerrail
      Contact( "CONV OVER SEL BIT" )
      Contact( "AL DOOR2 PRESS FAIL" )
      P_Trig( "AL1_6 TRIG" )
      S_Coil( "REQ AL1_6" )
   END_RUNG
   RUNG wire#powerrail
      Contact( "CONV OVER SEL BIT" )
      I_Contact( "AL DOOR2 PRESS FAIL" )
      { S7_Templates := "time_type := Time" } "IEC_Timer_0_DB_47".TP(pt := T#100MS, et =>)
      R_Coil( "REQ AL1_6" )
   END_RUNG
   RUNG wire#powerrail
      { S7_Templates := "[value_type := Int, str_type := String]" } VAL_STRG(IN := "HOUR", SIZE := 2, PREC := 0, FORMAT := 16#0000, P := 3, OUT => "REVAMP".ALM14)
   END_RUNG
   RUNG wire#powerrail
      { S7_Templates := "[value_type := Int, str_type := String]" } VAL_STRG(IN := "MINUTE", SIZE := 2, PREC := 0, FORMAT := 16#0000, P := 6, OUT => "REVAMP".ALM14)
   END_RUNG
   RUNG wire#powerrail
      { S7_Templates := "[value_type := Int, str_type := String]" } VAL_STRG(IN := "SECOND", SIZE := 2, PREC := 0, FORMAT := 16#0000, P := 9, OUT => "REVAMP".ALM14)
   END_RUNG
   // the same network as SCL:
   IF "START PV" AND "CONV OVER SEL BIT" THEN
       "SEND_PTP_DB_15"(REQ := "REQ AL1_6",   // SEND_PTP
                        PORT := "Local~CM_1241_(RS232)_1",
                        BUFFER := "REVAMP".ALM14,
                        DONE => "SEND_PTP_DB_15".DONE);
   END_IF;
   #_w1 := "CONV OVER SEL BIT" AND "AL DOOR2 PRESS FAIL";
   #_w2 := #_w1 AND NOT "AL1_6 TRIG";   // rising edge
   "AL1_6 TRIG" := #_w1;
   IF #_w2 THEN "REQ AL1_6" := TRUE; END_IF;
   "IEC_Timer_0_DB_47".TP(IN := "CONV OVER SEL BIT" AND NOT "AL DOOR2 PRESS FAIL", PT := T#100MS);
   IF "IEC_Timer_0_DB_47".Q THEN "REQ AL1_6" := FALSE; END_IF;
   VAL_STRG(IN := "HOUR", SIZE := 2, PREC := 0, FORMAT := 16#0000, P := 3, OUT => "REVAMP".ALM14);
   VAL_STRG(IN := "MINUTE", SIZE := 2, PREC := 0, FORMAT := 16#0000, P := 6, OUT => "REVAMP".ALM14);
   VAL_STRG(IN := "SECOND", SIZE := 2, PREC := 0, FORMAT := 16#0000, P := 9, OUT => "REVAMP".ALM14);
END_REGION

REGION Network 16
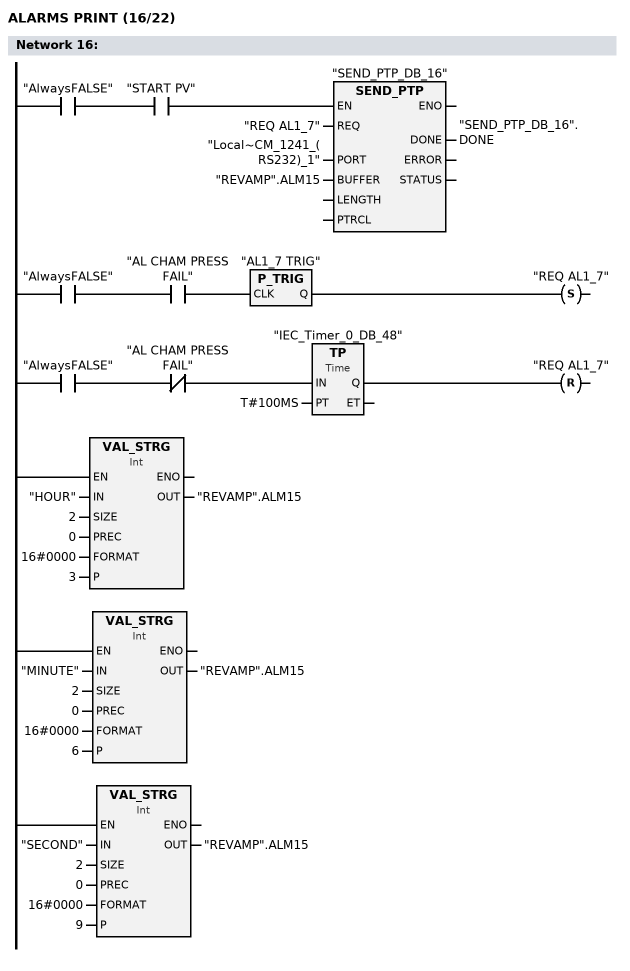
   RUNG wire#powerrail
      Contact( "AlwaysFALSE" )
      Contact( "START PV" )
      "SEND_PTP_DB_16".SEND_PTP(REQ := "REQ AL1_7", PORT := "Local~CM_1241_(RS232)_1", BUFFER := "REVAMP".ALM15, LENGTH :=, PTRCL :=, DONE => "SEND_PTP_DB_16".DONE, ERROR =>, STATUS =>)
   END_RUNG
   RUNG wire#powerrail
      Contact( "AlwaysFALSE" )
      Contact( "AL CHAM PRESS FAIL" )
      P_Trig( "AL1_7 TRIG" )
      S_Coil( "REQ AL1_7" )
   END_RUNG
   RUNG wire#powerrail
      Contact( "AlwaysFALSE" )
      I_Contact( "AL CHAM PRESS FAIL" )
      { S7_Templates := "time_type := Time" } "IEC_Timer_0_DB_48".TP(pt := T#100MS, et =>)
      R_Coil( "REQ AL1_7" )
   END_RUNG
   RUNG wire#powerrail
      { S7_Templates := "[value_type := Int, str_type := String]" } VAL_STRG(IN := "HOUR", SIZE := 2, PREC := 0, FORMAT := 16#0000, P := 3, OUT => "REVAMP".ALM15)
   END_RUNG
   RUNG wire#powerrail
      { S7_Templates := "[value_type := Int, str_type := String]" } VAL_STRG(IN := "MINUTE", SIZE := 2, PREC := 0, FORMAT := 16#0000, P := 6, OUT => "REVAMP".ALM15)
   END_RUNG
   RUNG wire#powerrail
      { S7_Templates := "[value_type := Int, str_type := String]" } VAL_STRG(IN := "SECOND", SIZE := 2, PREC := 0, FORMAT := 16#0000, P := 9, OUT => "REVAMP".ALM15)
   END_RUNG
   // the same network as SCL:
   IF "AlwaysFALSE" AND "START PV" THEN
       "SEND_PTP_DB_16"(REQ := "REQ AL1_7",   // SEND_PTP
                        PORT := "Local~CM_1241_(RS232)_1",
                        BUFFER := "REVAMP".ALM15,
                        DONE => "SEND_PTP_DB_16".DONE);
   END_IF;
   #_w1 := "AlwaysFALSE" AND "AL CHAM PRESS FAIL";
   #_w2 := #_w1 AND NOT "AL1_7 TRIG";   // rising edge
   "AL1_7 TRIG" := #_w1;
   IF #_w2 THEN "REQ AL1_7" := TRUE; END_IF;
   "IEC_Timer_0_DB_48".TP(IN := "AlwaysFALSE" AND NOT "AL CHAM PRESS FAIL", PT := T#100MS);
   IF "IEC_Timer_0_DB_48".Q THEN "REQ AL1_7" := FALSE; END_IF;
   VAL_STRG(IN := "HOUR", SIZE := 2, PREC := 0, FORMAT := 16#0000, P := 3, OUT => "REVAMP".ALM15);
   VAL_STRG(IN := "MINUTE", SIZE := 2, PREC := 0, FORMAT := 16#0000, P := 6, OUT => "REVAMP".ALM15);
   VAL_STRG(IN := "SECOND", SIZE := 2, PREC := 0, FORMAT := 16#0000, P := 9, OUT => "REVAMP".ALM15);
END_REGION

REGION Network 17
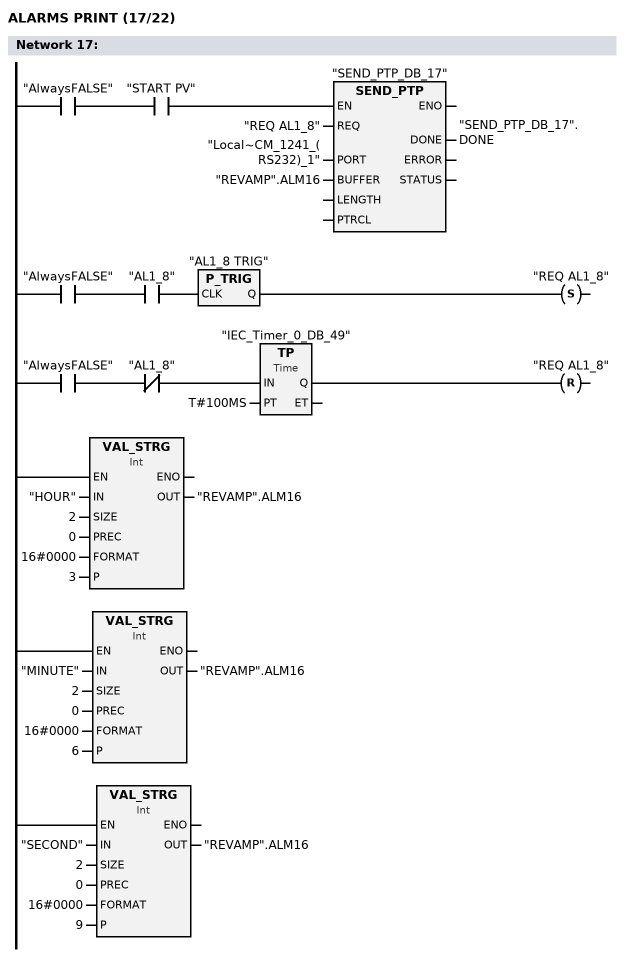
   RUNG wire#powerrail
      Contact( "AlwaysFALSE" )
      Contact( "START PV" )
      "SEND_PTP_DB_17".SEND_PTP(REQ := "REQ AL1_8", PORT := "Local~CM_1241_(RS232)_1", BUFFER := "REVAMP".ALM16, LENGTH :=, PTRCL :=, DONE => "SEND_PTP_DB_17".DONE, ERROR =>, STATUS =>)
   END_RUNG
   RUNG wire#powerrail
      Contact( "AlwaysFALSE" )
      Contact( "AL1_8" )
      P_Trig( "AL1_8 TRIG" )
      S_Coil( "REQ AL1_8" )
   END_RUNG
   RUNG wire#powerrail
      Contact( "AlwaysFALSE" )
      I_Contact( "AL1_8" )
      { S7_Templates := "time_type := Time" } "IEC_Timer_0_DB_49".TP(pt := T#100MS, et =>)
      R_Coil( "REQ AL1_8" )
   END_RUNG
   RUNG wire#powerrail
      { S7_Templates := "[value_type := Int, str_type := String]" } VAL_STRG(IN := "HOUR", SIZE := 2, PREC := 0, FORMAT := 16#0000, P := 3, OUT => "REVAMP".ALM16)
   END_RUNG
   RUNG wire#powerrail
      { S7_Templates := "[value_type := Int, str_type := String]" } VAL_STRG(IN := "MINUTE", SIZE := 2, PREC := 0, FORMAT := 16#0000, P := 6, OUT => "REVAMP".ALM16)
   END_RUNG
   RUNG wire#powerrail
      { S7_Templates := "[value_type := Int, str_type := String]" } VAL_STRG(IN := "SECOND", SIZE := 2, PREC := 0, FORMAT := 16#0000, P := 9, OUT => "REVAMP".ALM16)
   END_RUNG
   // the same network as SCL:
   IF "AlwaysFALSE" AND "START PV" THEN
       "SEND_PTP_DB_17"(REQ := "REQ AL1_8",   // SEND_PTP
                        PORT := "Local~CM_1241_(RS232)_1",
                        BUFFER := "REVAMP".ALM16,
                        DONE => "SEND_PTP_DB_17".DONE);
   END_IF;
   #_w1 := "AlwaysFALSE" AND "AL1_8";
   #_w2 := #_w1 AND NOT "AL1_8 TRIG";   // rising edge
   "AL1_8 TRIG" := #_w1;
   IF #_w2 THEN "REQ AL1_8" := TRUE; END_IF;
   "IEC_Timer_0_DB_49".TP(IN := "AlwaysFALSE" AND NOT "AL1_8", PT := T#100MS);
   IF "IEC_Timer_0_DB_49".Q THEN "REQ AL1_8" := FALSE; END_IF;
   VAL_STRG(IN := "HOUR", SIZE := 2, PREC := 0, FORMAT := 16#0000, P := 3, OUT => "REVAMP".ALM16);
   VAL_STRG(IN := "MINUTE", SIZE := 2, PREC := 0, FORMAT := 16#0000, P := 6, OUT => "REVAMP".ALM16);
   VAL_STRG(IN := "SECOND", SIZE := 2, PREC := 0, FORMAT := 16#0000, P := 9, OUT => "REVAMP".ALM16);
END_REGION

REGION Network 18
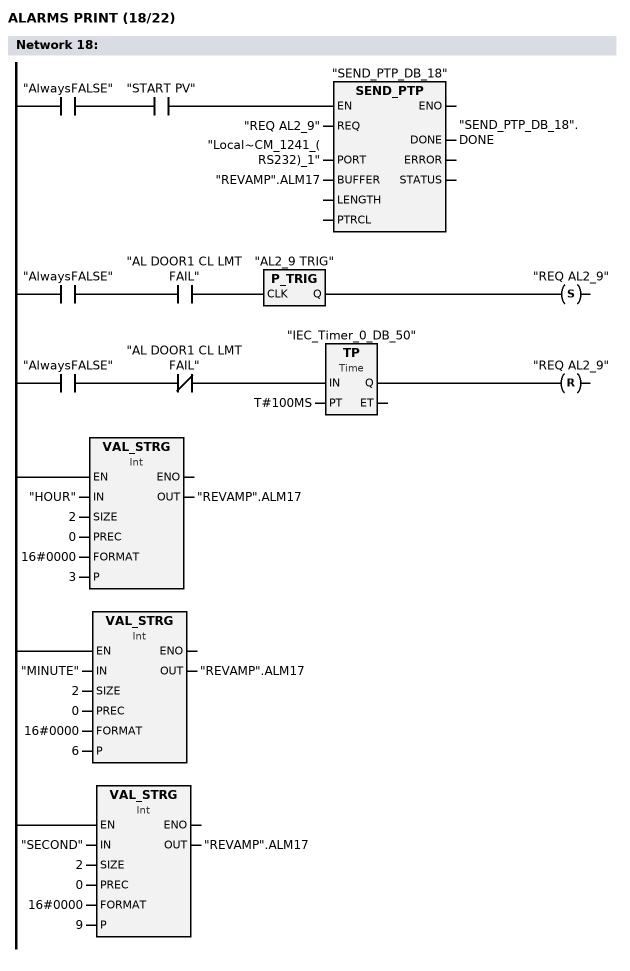
   RUNG wire#powerrail
      Contact( "AlwaysFALSE" )
      Contact( "START PV" )
      "SEND_PTP_DB_18".SEND_PTP(REQ := "REQ AL2_9", PORT := "Local~CM_1241_(RS232)_1", BUFFER := "REVAMP".ALM17, LENGTH :=, PTRCL :=, DONE => "SEND_PTP_DB_18".DONE, ERROR =>, STATUS =>)
   END_RUNG
   RUNG wire#powerrail
      Contact( "AlwaysFALSE" )
      Contact( "AL DOOR1 CL LMT FAIL" )
      P_Trig( "AL2_9 TRIG" )
      S_Coil( "REQ AL2_9" )
   END_RUNG
   RUNG wire#powerrail
      Contact( "AlwaysFALSE" )
      I_Contact( "AL DOOR1 CL LMT FAIL" )
      { S7_Templates := "time_type := Time" } "IEC_Timer_0_DB_50".TP(pt := T#100MS, et =>)
      R_Coil( "REQ AL2_9" )
   END_RUNG
   RUNG wire#powerrail
      { S7_Templates := "[value_type := Int, str_type := String]" } VAL_STRG(IN := "HOUR", SIZE := 2, PREC := 0, FORMAT := 16#0000, P := 3, OUT => "REVAMP".ALM17)
   END_RUNG
   RUNG wire#powerrail
      { S7_Templates := "[value_type := Int, str_type := String]" } VAL_STRG(IN := "MINUTE", SIZE := 2, PREC := 0, FORMAT := 16#0000, P := 6, OUT => "REVAMP".ALM17)
   END_RUNG
   RUNG wire#powerrail
      { S7_Templates := "[value_type := Int, str_type := String]" } VAL_STRG(IN := "SECOND", SIZE := 2, PREC := 0, FORMAT := 16#0000, P := 9, OUT => "REVAMP".ALM17)
   END_RUNG
   // the same network as SCL:
   IF "AlwaysFALSE" AND "START PV" THEN
       "SEND_PTP_DB_18"(REQ := "REQ AL2_9",   // SEND_PTP
                        PORT := "Local~CM_1241_(RS232)_1",
                        BUFFER := "REVAMP".ALM17,
                        DONE => "SEND_PTP_DB_18".DONE);
   END_IF;
   #_w1 := "AlwaysFALSE" AND "AL DOOR1 CL LMT FAIL";
   #_w2 := #_w1 AND NOT "AL2_9 TRIG";   // rising edge
   "AL2_9 TRIG" := #_w1;
   IF #_w2 THEN "REQ AL2_9" := TRUE; END_IF;
   "IEC_Timer_0_DB_50".TP(IN := "AlwaysFALSE" AND NOT "AL DOOR1 CL LMT FAIL", PT := T#100MS);
   IF "IEC_Timer_0_DB_50".Q THEN "REQ AL2_9" := FALSE; END_IF;
   VAL_STRG(IN := "HOUR", SIZE := 2, PREC := 0, FORMAT := 16#0000, P := 3, OUT => "REVAMP".ALM17);
   VAL_STRG(IN := "MINUTE", SIZE := 2, PREC := 0, FORMAT := 16#0000, P := 6, OUT => "REVAMP".ALM17);
   VAL_STRG(IN := "SECOND", SIZE := 2, PREC := 0, FORMAT := 16#0000, P := 9, OUT => "REVAMP".ALM17);
END_REGION

REGION Network 19
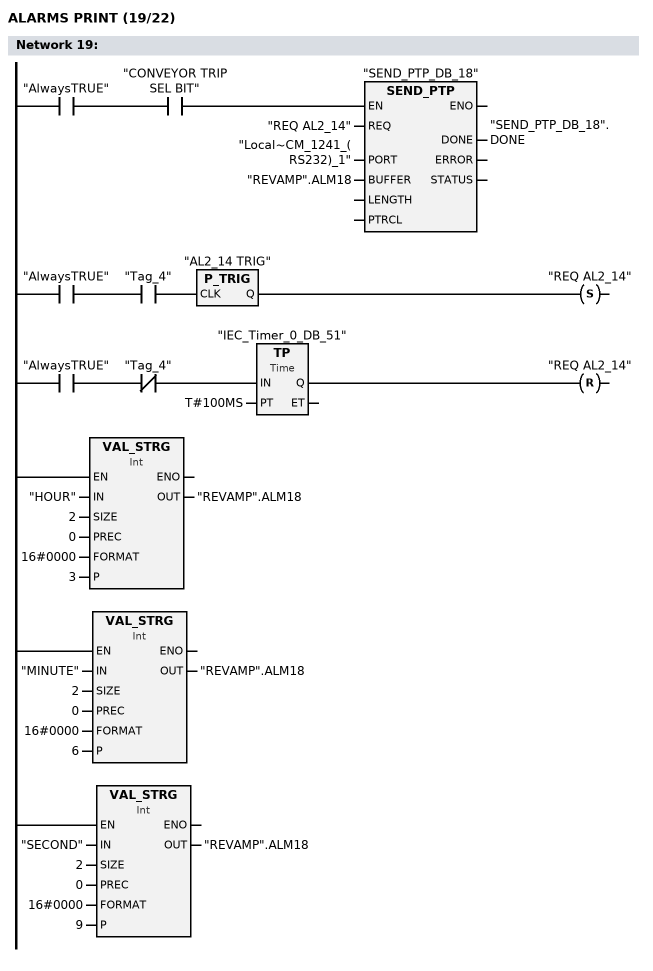
   RUNG wire#powerrail
      Contact( "AlwaysTRUE" )
      Contact( "CONVEYOR TRIP SEL BIT" )
      "SEND_PTP_DB_18".SEND_PTP(REQ := "REQ AL2_14", PORT := "Local~CM_1241_(RS232)_1", BUFFER := "REVAMP".ALM18, LENGTH :=, PTRCL :=, DONE => "SEND_PTP_DB_18".DONE, ERROR =>, STATUS =>)
   END_RUNG
   RUNG wire#powerrail
      Contact( "AlwaysTRUE" )
      Contact( "Tag_4" )
      P_Trig( "AL2_14 TRIG" )
      S_Coil( "REQ AL2_14" )
   END_RUNG
   RUNG wire#powerrail
      Contact( "AlwaysTRUE" )
      I_Contact( "Tag_4" )
      { S7_Templates := "time_type := Time" } "IEC_Timer_0_DB_51".TP(pt := T#100MS, et =>)
      R_Coil( "REQ AL2_14" )
   END_RUNG
   RUNG wire#powerrail
      { S7_Templates := "[value_type := Int, str_type := String]" } VAL_STRG(IN := "HOUR", SIZE := 2, PREC := 0, FORMAT := 16#0000, P := 3, OUT => "REVAMP".ALM18)
   END_RUNG
   RUNG wire#powerrail
      { S7_Templates := "[value_type := Int, str_type := String]" } VAL_STRG(IN := "MINUTE", SIZE := 2, PREC := 0, FORMAT := 16#0000, P := 6, OUT => "REVAMP".ALM18)
   END_RUNG
   RUNG wire#powerrail
      { S7_Templates := "[value_type := Int, str_type := String]" } VAL_STRG(IN := "SECOND", SIZE := 2, PREC := 0, FORMAT := 16#0000, P := 9, OUT => "REVAMP".ALM18)
   END_RUNG
   // the same network as SCL:
   IF "AlwaysTRUE" AND "CONVEYOR TRIP SEL BIT" THEN
       "SEND_PTP_DB_18"(REQ := "REQ AL2_14",   // SEND_PTP
                        PORT := "Local~CM_1241_(RS232)_1",
                        BUFFER := "REVAMP".ALM18,
                        DONE => "SEND_PTP_DB_18".DONE);
   END_IF;
   #_w1 := "AlwaysTRUE" AND "Tag_4";
   #_w2 := #_w1 AND NOT "AL2_14 TRIG";   // rising edge
   "AL2_14 TRIG" := #_w1;
   IF #_w2 THEN "REQ AL2_14" := TRUE; END_IF;
   "IEC_Timer_0_DB_51".TP(IN := "AlwaysTRUE" AND NOT "Tag_4", PT := T#100MS);
   IF "IEC_Timer_0_DB_51".Q THEN "REQ AL2_14" := FALSE; END_IF;
   VAL_STRG(IN := "HOUR", SIZE := 2, PREC := 0, FORMAT := 16#0000, P := 3, OUT => "REVAMP".ALM18);
   VAL_STRG(IN := "MINUTE", SIZE := 2, PREC := 0, FORMAT := 16#0000, P := 6, OUT => "REVAMP".ALM18);
   VAL_STRG(IN := "SECOND", SIZE := 2, PREC := 0, FORMAT := 16#0000, P := 9, OUT => "REVAMP".ALM18);
END_REGION

REGION Network 20
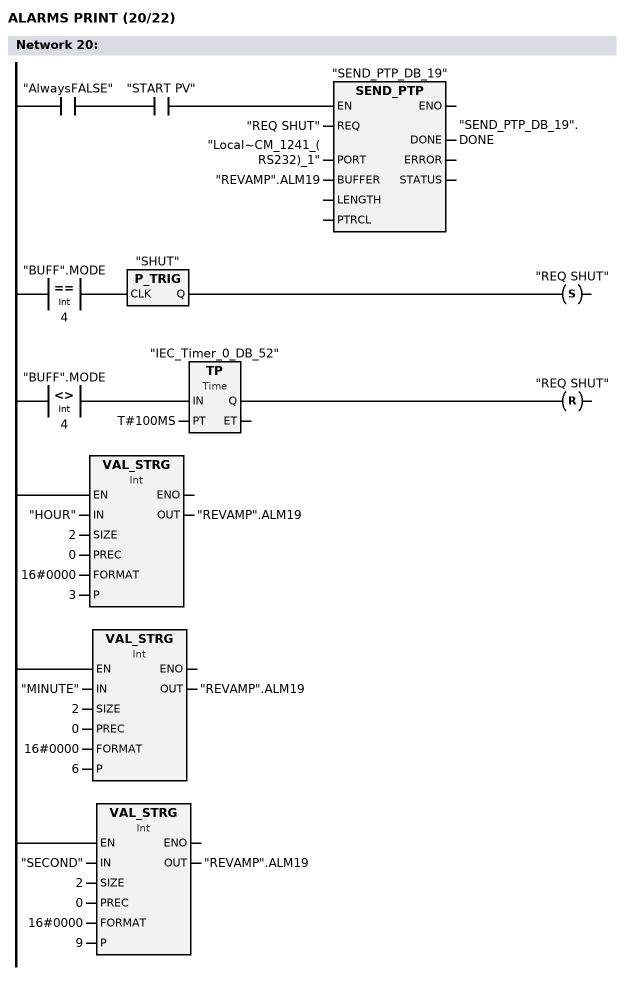
   RUNG wire#powerrail
      Contact( "AlwaysFALSE" )
      Contact( "START PV" )
      "SEND_PTP_DB_19".SEND_PTP(REQ := "REQ SHUT", PORT := "Local~CM_1241_(RS232)_1", BUFFER := "REVAMP".ALM19, LENGTH :=, PTRCL :=, DONE => "SEND_PTP_DB_19".DONE, ERROR =>, STATUS =>)
   END_RUNG
   RUNG wire#powerrail
      { S7_Templates := "SrcType := Int" } EQ_Contact(in1 := "BUFF".MODE, in2 := 4)
      P_Trig( "SHUT" )
      S_Coil( "REQ SHUT" )
   END_RUNG
   RUNG wire#powerrail
      { S7_Templates := "SrcType := Int" } NE_Contact(in1 := "BUFF".MODE, in2 := 4)
      { S7_Templates := "time_type := Time" } "IEC_Timer_0_DB_52".TP(pt := T#100MS, et =>)
      R_Coil( "REQ SHUT" )
   END_RUNG
   RUNG wire#powerrail
      { S7_Templates := "[value_type := Int, str_type := String]" } VAL_STRG(IN := "HOUR", SIZE := 2, PREC := 0, FORMAT := 16#0000, P := 3, OUT => "REVAMP".ALM19)
   END_RUNG
   RUNG wire#powerrail
      { S7_Templates := "[value_type := Int, str_type := String]" } VAL_STRG(IN := "MINUTE", SIZE := 2, PREC := 0, FORMAT := 16#0000, P := 6, OUT => "REVAMP".ALM19)
   END_RUNG
   RUNG wire#powerrail
      { S7_Templates := "[value_type := Int, str_type := String]" } VAL_STRG(IN := "SECOND", SIZE := 2, PREC := 0, FORMAT := 16#0000, P := 9, OUT => "REVAMP".ALM19)
   END_RUNG
   // the same network as SCL:
   IF "AlwaysFALSE" AND "START PV" THEN
       "SEND_PTP_DB_19"(REQ := "REQ SHUT",   // SEND_PTP
                        PORT := "Local~CM_1241_(RS232)_1",
                        BUFFER := "REVAMP".ALM19,
                        DONE => "SEND_PTP_DB_19".DONE);
   END_IF;
   #_w1 := "BUFF".MODE = 4;
   #_w2 := #_w1 AND NOT "SHUT";   // rising edge
   "SHUT" := #_w1;
   IF #_w2 THEN "REQ SHUT" := TRUE; END_IF;
   "IEC_Timer_0_DB_52".TP(IN := "BUFF".MODE <> 4, PT := T#100MS);
   IF "IEC_Timer_0_DB_52".Q THEN "REQ SHUT" := FALSE; END_IF;
   VAL_STRG(IN := "HOUR", SIZE := 2, PREC := 0, FORMAT := 16#0000, P := 3, OUT => "REVAMP".ALM19);
   VAL_STRG(IN := "MINUTE", SIZE := 2, PREC := 0, FORMAT := 16#0000, P := 6, OUT => "REVAMP".ALM19);
   VAL_STRG(IN := "SECOND", SIZE := 2, PREC := 0, FORMAT := 16#0000, P := 9, OUT => "REVAMP".ALM19);
END_REGION

REGION Network 21
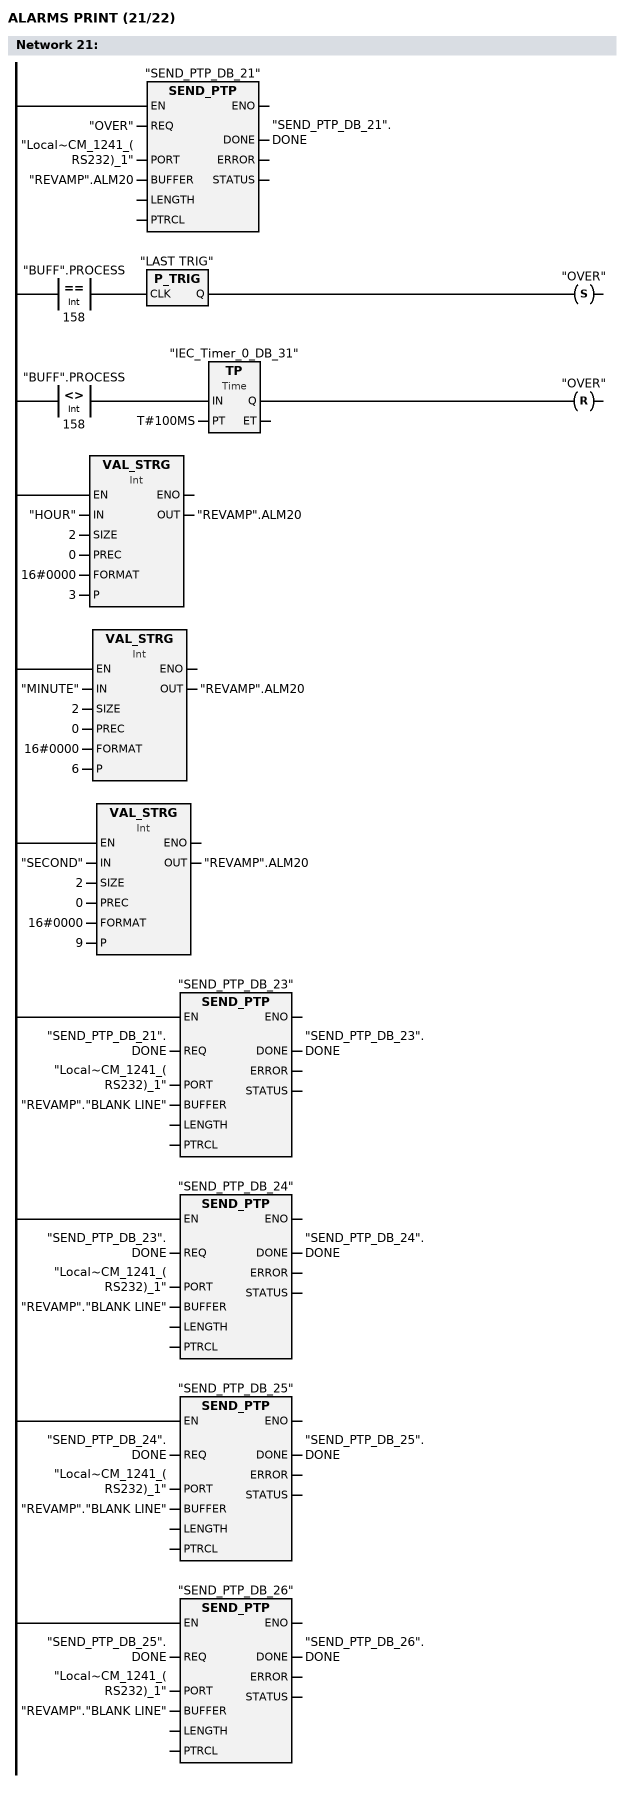
   RUNG wire#powerrail
      "SEND_PTP_DB_21".SEND_PTP(REQ := "OVER", PORT := "Local~CM_1241_(RS232)_1", BUFFER := "REVAMP".ALM20, LENGTH :=, PTRCL :=, DONE => "SEND_PTP_DB_21".DONE, ERROR =>, STATUS =>)
   END_RUNG
   RUNG wire#powerrail
      { S7_Templates := "SrcType := Int" } EQ_Contact(in1 := "BUFF".PROCESS, in2 := 158)
      P_Trig( "LAST TRIG" )
      S_Coil( "OVER" )
   END_RUNG
   RUNG wire#powerrail
      { S7_Templates := "SrcType := Int" } NE_Contact(in1 := "BUFF".PROCESS, in2 := 158)
      { S7_Templates := "time_type := Time" } "IEC_Timer_0_DB_31".TP(pt := T#100MS, et =>)
      R_Coil( "OVER" )
   END_RUNG
   RUNG wire#powerrail
      { S7_Templates := "[value_type := Int, str_type := String]" } VAL_STRG(IN := "HOUR", SIZE := 2, PREC := 0, FORMAT := 16#0000, P := 3, OUT => "REVAMP".ALM20)
   END_RUNG
   RUNG wire#powerrail
      { S7_Templates := "[value_type := Int, str_type := String]" } VAL_STRG(IN := "MINUTE", SIZE := 2, PREC := 0, FORMAT := 16#0000, P := 6, OUT => "REVAMP".ALM20)
   END_RUNG
   RUNG wire#powerrail
      { S7_Templates := "[value_type := Int, str_type := String]" } VAL_STRG(IN := "SECOND", SIZE := 2, PREC := 0, FORMAT := 16#0000, P := 9, OUT => "REVAMP".ALM20)
   END_RUNG
   RUNG wire#powerrail
      "SEND_PTP_DB_23".SEND_PTP(REQ := "SEND_PTP_DB_21".DONE, PORT := "Local~CM_1241_(RS232)_1", BUFFER := "REVAMP"."BLANK LINE", LENGTH :=, PTRCL :=, DONE => "SEND_PTP_DB_23".DONE, ERROR =>, STATUS =>)
   END_RUNG
   RUNG wire#powerrail
      "SEND_PTP_DB_24".SEND_PTP(REQ := "SEND_PTP_DB_23".DONE, PORT := "Local~CM_1241_(RS232)_1", BUFFER := "REVAMP"."BLANK LINE", LENGTH :=, PTRCL :=, DONE => "SEND_PTP_DB_24".DONE, ERROR =>, STATUS =>)
   END_RUNG
   RUNG wire#powerrail
      "SEND_PTP_DB_25".SEND_PTP(REQ := "SEND_PTP_DB_24".DONE, PORT := "Local~CM_1241_(RS232)_1", BUFFER := "REVAMP"."BLANK LINE", LENGTH :=, PTRCL :=, DONE => "SEND_PTP_DB_25".DONE, ERROR =>, STATUS =>)
   END_RUNG
   RUNG wire#powerrail
      "SEND_PTP_DB_26".SEND_PTP(REQ := "SEND_PTP_DB_25".DONE, PORT := "Local~CM_1241_(RS232)_1", BUFFER := "REVAMP"."BLANK LINE", LENGTH :=, PTRCL :=, DONE => "SEND_PTP_DB_26".DONE, ERROR =>, STATUS =>)
   END_RUNG
   // the same network as SCL:
   "SEND_PTP_DB_21"(REQ := "OVER",   // SEND_PTP
                    PORT := "Local~CM_1241_(RS232)_1",
                    BUFFER := "REVAMP".ALM20,
                    DONE => "SEND_PTP_DB_21".DONE);
   #_w1 := "BUFF".PROCESS = 158;
   #_w2 := #_w1 AND NOT "LAST TRIG";   // rising edge
   "LAST TRIG" := #_w1;
   IF #_w2 THEN "OVER" := TRUE; END_IF;
   "IEC_Timer_0_DB_31".TP(IN := "BUFF".PROCESS <> 158, PT := T#100MS);
   IF "IEC_Timer_0_DB_31".Q THEN "OVER" := FALSE; END_IF;
   VAL_STRG(IN := "HOUR", SIZE := 2, PREC := 0, FORMAT := 16#0000, P := 3, OUT => "REVAMP".ALM20);
   VAL_STRG(IN := "MINUTE", SIZE := 2, PREC := 0, FORMAT := 16#0000, P := 6, OUT => "REVAMP".ALM20);
   VAL_STRG(IN := "SECOND", SIZE := 2, PREC := 0, FORMAT := 16#0000, P := 9, OUT => "REVAMP".ALM20);
   "SEND_PTP_DB_23"(REQ := "SEND_PTP_DB_21".DONE,   // SEND_PTP
                    PORT := "Local~CM_1241_(RS232)_1",
                    BUFFER := "REVAMP"."BLANK LINE",
                    DONE => "SEND_PTP_DB_23".DONE);
   "SEND_PTP_DB_24"(REQ := "SEND_PTP_DB_23".DONE,   // SEND_PTP
                    PORT := "Local~CM_1241_(RS232)_1",
                    BUFFER := "REVAMP"."BLANK LINE",
                    DONE => "SEND_PTP_DB_24".DONE);
   "SEND_PTP_DB_25"(REQ := "SEND_PTP_DB_24".DONE,   // SEND_PTP
                    PORT := "Local~CM_1241_(RS232)_1",
                    BUFFER := "REVAMP"."BLANK LINE",
                    DONE => "SEND_PTP_DB_25".DONE);
   "SEND_PTP_DB_26"(REQ := "SEND_PTP_DB_25".DONE,   // SEND_PTP
                    PORT := "Local~CM_1241_(RS232)_1",
                    BUFFER := "REVAMP"."BLANK LINE",
                    DONE => "SEND_PTP_DB_26".DONE);
END_REGION

REGION Network 22
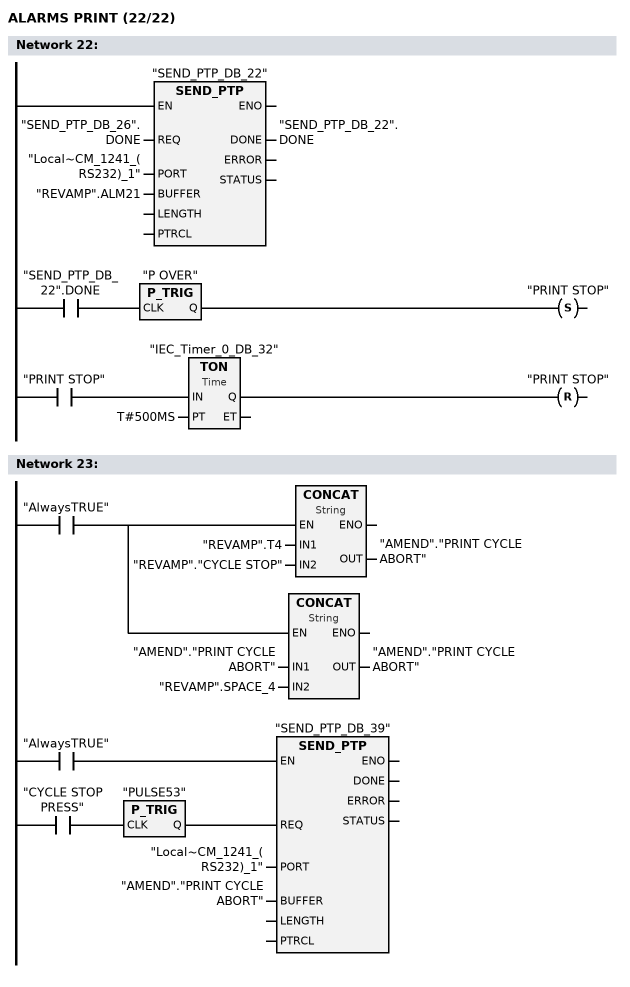
   RUNG wire#powerrail
      "SEND_PTP_DB_22".SEND_PTP(REQ := "SEND_PTP_DB_26".DONE, PORT := "Local~CM_1241_(RS232)_1", BUFFER := "REVAMP".ALM21, LENGTH :=, PTRCL :=, DONE => "SEND_PTP_DB_22".DONE, ERROR =>, STATUS =>)
   END_RUNG
   RUNG wire#powerrail
      Contact( "SEND_PTP_DB_22".DONE )
      P_Trig( "P OVER" )
      S_Coil( "PRINT STOP" )
   END_RUNG
   RUNG wire#powerrail
      Contact( "PRINT STOP" )
      { S7_Templates := "time_type := Time" } "IEC_Timer_0_DB_32".TON(pt := T#500MS, et =>)
      R_Coil( "PRINT STOP" )
   END_RUNG
   // the same network as SCL:
   "SEND_PTP_DB_22"(REQ := "SEND_PTP_DB_26".DONE,   // SEND_PTP
                    PORT := "Local~CM_1241_(RS232)_1",
                    BUFFER := "REVAMP".ALM21,
                    DONE => "SEND_PTP_DB_22".DONE);
   #_w1 := "SEND_PTP_DB_22".DONE AND NOT "P OVER";   // rising edge
   "P OVER" := "SEND_PTP_DB_22".DONE;
   IF #_w1 THEN "PRINT STOP" := TRUE; END_IF;
   "IEC_Timer_0_DB_32".TON(IN := "PRINT STOP", PT := T#500MS);
   IF "IEC_Timer_0_DB_32".Q THEN "PRINT STOP" := FALSE; END_IF;
END_REGION

REGION Network 23
   RUNG wire#powerrail
      Contact( "AlwaysTRUE" )
      wire#w1
      { S7_Templates := "[card := 2, str_type := String]" } CONCAT(IN1 := "REVAMP".T4, IN2 := "REVAMP"."CYCLE STOP", OUT => "AMEND"."PRINT CYCLE ABORT")
   END_RUNG
   RUNG wire#w1
      { S7_Templates := "[card := 2, str_type := String]" } CONCAT(IN1 := "AMEND"."PRINT CYCLE ABORT", IN2 := "REVAMP".SPACE_4, OUT => "AMEND"."PRINT CYCLE ABORT")
   END_RUNG
   RUNG wire#powerrail
      Contact( "AlwaysTRUE" )
      "SEND_PTP_DB_39".SEND_PTP(REQ := wire#w2, PORT := "Local~CM_1241_(RS232)_1", BUFFER := "AMEND"."PRINT CYCLE ABORT", LENGTH :=, PTRCL :=, DONE =>, ERROR =>, STATUS =>)
   END_RUNG
   RUNG wire#powerrail
      Contact( "CYCLE STOP PRESS" )
      P_Trig( "PULSE53" )
   END_RUNG wire#w2
   // the same network as SCL:
   #_w1 := "AlwaysTRUE";
   IF #_w1 THEN
       CONCAT(IN1 := "REVAMP".T4, IN2 := "REVAMP"."CYCLE STOP", OUT => "AMEND"."PRINT CYCLE ABORT");
       CONCAT(IN1 := "AMEND"."PRINT CYCLE ABORT", IN2 := "REVAMP".SPACE_4, OUT => "AMEND"."PRINT CYCLE ABORT");
   END_IF;
   #_w2 := "CYCLE STOP PRESS" AND NOT "PULSE53";   // rising edge
   "PULSE53" := "CYCLE STOP PRESS";
   IF "AlwaysTRUE" THEN
       "SEND_PTP_DB_39"(REQ := #_w2, PORT := "Local~CM_1241_(RS232)_1", BUFFER := "AMEND"."PRINT CYCLE ABORT");   // SEND_PTP
   END_IF;
END_REGION
END_FUNCTION
